LIN {X 0,Y 333.644,Z 264.427,A -85,B 0,C 180,E1 -14639.633,E2 -14639.633} C_VEL
LIN {X 0,Y 333.689,Z 264.417,A -85,B 0,C 180,E1 -14642.397,E2 -14642.397} C_VEL
LIN {X 0,Y 333.704,Z 264.416,A -85,B 0,C 180,E1 -14645.09,E2 -14645.09} C_VEL
LIN {X 0,Y 333.673,Z 264.443,A -85,B 0,C 180,E1 -14648.774,E2 -14648.774} C_VEL
LIN {X 0,Y 334.576,Z 267.116,A -85,B 0,C 180,E1 -14648.985,E2 -14648.985} C_VEL
LIN {X 0,Y 336.917,Z 269.949,A -85,B 0,C 180,E1 -14649.425,E2 -14649.425} C_VEL
LIN {X 0,Y 339.171,Z 273.256,A -85,B 0,C 180,E1 -14649.871,E2 -14649.871} C_VEL
LIN {X 0,Y 340.664,Z 274.981,A -85,B 0,C 180,E1 -14650.162,E2 -14650.162} C_VEL
LIN {X 0,Y 343.625,Z 278.711,A -85,B 0,C 180,E1 -14650.768,E2 -14650.768} C_VEL
LIN {X 0,Y 345.334,Z 280.75,A -85,B 0,C 180,E1 -14651.122,E2 -14651.122} C_VEL
LIN {X 0,Y 348.82,Z 284.693,A -85,B 0,C 180,E1 -14651.877,E2 -14651.877} C_VEL
LIN {X 0,Y 353.769,Z 290.158,A -85,B 0,C 180,E1 -14653.004,E2 -14653.004} C_VEL
LIN {X 0,Y 355.969,Z 292.267,A -85,B 0,C 180,E1 -14653.529,E2 -14653.529} C_VEL
LIN {X 0,Y 359.569,Z 296.096,A -85,B 0,C 180,E1 -14654.442,E2 -14654.442} C_VEL
LIN {X 0,Y 362.57,Z 298.711,A -85,B 0,C 180,E1 -14655.235,E2 -14655.235} C_VEL
LIN {X 0,Y 366.124,Z 302.39,A -85,B 0,C 180,E1 -14656.282,E2 -14656.282} C_VEL
LIN {X 0,Y 370.169,Z 305.771,A -85,B 0,C 180,E1 -14657.554,E2 -14657.554} C_VEL
LIN {X 0,Y 373.465,Z 309.144,A -85,B 0,C 180,E1 -14658.767,E2 -14658.767} C_VEL
LIN {X 0,Y 377.002,Z 311.663,A -85,B 0,C 180,E1 -14660.138,E2 -14660.138} C_VEL
LIN {X 0,Y 378.672,Z 312.756,A -85,B 0,C 180,E1 -14660.864,E2 -14660.864} C_VEL
LIN {X 0,Y 381.373,Z 315.868,A -85,B 0,C 180,E1 -14662.35,E2 -14662.35} C_VEL
LIN {X 0,Y 383.817,Z 317.899,A -85,B 0,C 180,E1 -14663.899,E2 -14663.899} C_VEL
LIN {X 0,Y 385.982,Z 319.066,A -85,B 0,C 180,E1 -14665.59,E2 -14665.59} C_VEL
LIN {X 0,Y 387.241,Z 319.408,A -85,B 0,C 180,E1 -14666.879,E2 -14666.879} C_VEL
LIN {X 0,Y 387.946,Z 319.576,A -85,B 0,C 180,E1 -14667.924,E2 -14667.924} C_VEL
LIN {X 0,Y 388.385,Z 319.645,A -85,B 0,C 180,E1 -14668.963,E2 -14668.963} C_VEL
LIN {X 0,Y 388.544,Z 319.673,A -85,B 0,C 180,E1 -14670,E2 -14670} C_VEL
LIN {X 0,Y 388.383,Z 319.645,A -85,B 0,C 180,E1 -14671.037,E2 -14671.037} C_VEL
LIN {X 0,Y 387.236,Z 319.4,A -85,B 0,C 180,E1 -14673.121,E2 -14673.121} C_VEL
LIN {X 0,Y 385.289,Z 318.79,A -85,B 0,C 180,E1 -14674.995,E2 -14674.995} C_VEL
LIN {X 0,Y 382.667,Z 317.06,A -85,B 0,C 180,E1 -14676.858,E2 -14676.858} C_VEL
LIN {X 0,Y 379.94,Z 314.347,A -85,B 0,C 180,E1 -14678.455,E2 -14678.455} C_VEL
LIN {X 0,Y 378.086,Z 312.243,A -85,B 0,C 180,E1 -14679.384,E2 -14679.384} C_VEL
LIN {X 0,Y 374.748,Z 310.2,A -85,B 0,C 180,E1 -14680.732,E2 -14680.732} C_VEL
LIN {X 0,Y 371.26,Z 307.035,A -85,B 0,C 180,E1 -14682.053,E2 -14682.053} C_VEL
LIN {X 0,Y 368.774,Z 304.446,A -85,B 0,C 180,E1 -14682.914,E2 -14682.914} C_VEL
LIN {X 0,Y 364.898,Z 301.318,A -85,B 0,C 180,E1 -14684.081,E2 -14684.081} C_VEL
LIN {X 0,Y 361.298,Z 297.476,A -85,B 0,C 180,E1 -14685.115,E2 -14685.115} C_VEL
LIN {X 0,Y 357.215,Z 293.734,A -85,B 0,C 180,E1 -14686.17,E2 -14686.17} C_VEL
LIN {X 0,Y 354.441,Z 290.752,A -85,B 0,C 180,E1 -14686.836,E2 -14686.836} C_VEL
LIN {X 0,Y 350.86,Z 287.08,A -85,B 0,C 180,E1 -14687.662,E2 -14687.662} C_VEL
LIN {X 0,Y 348.59,Z 284.464,A -85,B 0,C 180,E1 -14688.174,E2 -14688.174} C_VEL
LIN {X 0,Y 345.334,Z 280.748,A -85,B 0,C 180,E1 -14688.878,E2 -14688.878} C_VEL
LIN {X 0,Y 343.74,Z 278.843,A -85,B 0,C 180,E1 -14689.208,E2 -14689.208} C_VEL
LIN {X 0,Y 340.623,Z 274.921,A -85,B 0,C 180,E1 -14689.846,E2 -14689.846} C_VEL
LIN {X 0,Y 337.257,Z 270.639,A -85,B 0,C 180,E1 -14690.505,E2 -14690.505} C_VEL
LIN {X 0,Y 336.338,Z 269.129,A -85,B 0,C 180,E1 -14690.687,E2 -14690.687} C_VEL
LIN {X 0,Y 334.367,Z 266.73,A -85,B 0,C 180,E1 -14691.058,E2 -14691.058} C_VEL
LIN {X 0,Y 333.667,Z 264.421,A -85,B 0,C 180,E1 -14691.261,E2 -14691.261} C_VEL
LIN {X 0,Y 333.674,Z 264.419,A -85,B 0,C 180,E1 -14695.108,E2 -14695.108} C_VEL
LIN {X 0,Y 333.667,Z 264.421,A -85,B 0,C 180,E1 -14697.814,E2 -14697.814} C_VEL
LIN {X 0,Y 333.644,Z 264.427,A -85,B 0,C 180,E1 -14700.367,E2 -14700.367} C_VEL
LIN {X 0,Y 333.634,Z 264.424,A -85,B 0,C 180,E1 -14704.779,E2 -14704.779} C_VEL
LIN {X 0,Y 333.631,Z 264.424,A -85,B 0,C 180,E1 -14708.809,E2 -14708.809} C_VEL
LIN {X 0,Y 333.657,Z 264.421,A -85,B 0,C 180,E1 -14712.519,E2 -14712.519} C_VEL
LIN {X 0,Y 333.687,Z 264.421,A -85,B 0,C 180,E1 -14715.983,E2 -14715.983} C_VEL
LIN {X 0,Y 333.662,Z 264.421,A -85,B 0,C 180,E1 -14719.311,E2 -14719.311} C_VEL
LIN {X 0,Y 333.628,Z 264.425,A -85,B 0,C 180,E1 -14723.175,E2 -14723.175} C_VEL
LIN {X 0,Y 333.604,Z 264.427,A -85,B 0,C 180,E1 -14726.799,E2 -14726.799} C_VEL
LIN {X 0,Y 333.649,Z 264.423,A -85,B 0,C 180,E1 -14731.032,E2 -14731.032} C_VEL
LIN {X 0,Y 333.681,Z 264.417,A -85,B 0,C 180,E1 -14734.672,E2 -14734.672} C_VEL
LIN {X 0,Y 333.639,Z 264.423,A -85,B 0,C 180,E1 -14737.945,E2 -14737.945} C_VEL
LIN {X 0,Y 333.622,Z 264.423,A -85,B 0,C 180,E1 -14739.904,E2 -14739.904} C_VEL
LIN {X 0,Y 332.986,Z 264.507,A -85,B 0,C 180,E1 -14740.912,E2 -14740.912} C_VEL
LIN {X 0,Y 330.181,Z 264.858,A -85,B 0,C 180,E1 -14742.552,E2 -14742.552} C_VEL
LIN {X 0,Y 327.805,Z 265.156,A -85,B 0,C 180,E1 -14743.881,E2 -14743.881} C_VEL
LIN {X 0,Y 326.806,Z 265.278,A -85,B 0,C 180,E1 -14744.909,E2 -14744.909} C_VEL
LIN {X 0,Y 326.736,Z 265.285,A -85,B 0,C 180,E1 -14745.257,E2 -14745.257} C_VEL
LIN {X 0,Y 326.741,Z 265.286,A -85,B 0,C 180,E1 -14748.846,E2 -14748.846} C_VEL
LIN {X 0,Y 326.925,Z 265.261,A -85,B 0,C 180,E1 -14752.597,E2 -14752.597} C_VEL
LIN {X 0,Y 326.754,Z 265.282,A -85,B 0,C 180,E1 -14755.072,E2 -14755.072} C_VEL
LIN {X 0,Y 327.033,Z 265.241,A -85,B 0,C 180,E1 -14757.544,E2 -14757.544} C_VEL
LIN {X 0,Y 327.15,Z 265.228,A -85,B 0,C 180,E1 -14760.007,E2 -14760.007} C_VEL
LIN {X 0,Y 327.005,Z 265.252,A -85,B 0,C 180,E1 -14762.471,E2 -14762.471} C_VEL
LIN {X 0,Y 326.948,Z 265.258,A -85,B 0,C 180,E1 -14766.177,E2 -14766.177} C_VEL
LIN {X 0,Y 326.781,Z 265.278,A -85,B 0,C 180,E1 -14769.914,E2 -14769.914} C_VEL
LIN {X 0,Y 326.76,Z 265.28,A -85,B 0,C 180,E1 -14773.692,E2 -14773.692} C_VEL
LIN {X 0,Y 326.666,Z 265.292,A -85,B 0,C 180,E1 -14777.536,E2 -14777.536} C_VEL
LIN {X 0,Y 326.619,Z 265.298,A -85,B 0,C 180,E1 -14781.463,E2 -14781.463} C_VEL
LIN {X 0,Y 326.611,Z 265.3,A -85,B 0,C 180,E1 -14785.497,E2 -14785.497} C_VEL
LIN {X 0,Y 326.624,Z 265.3,A -85,B 0,C 180,E1 -14789.669,E2 -14789.669} C_VEL
LIN {X 0,Y 326.627,Z 265.299,A -85,B 0,C 180,E1 -14792.951,E2 -14792.951} C_VEL
LIN {X 0,Y 326.695,Z 265.648,A -85,B 0,C 180,E1 -14795.516,E2 -14795.516} C_VEL
LIN {X 0,Y 327.028,Z 268.288,A -85,B 0,C 180,E1 -14799.318,E2 -14799.318} C_VEL
LIN {X 0,Y 327.449,Z 271.2,A -85,B 0,C 180,E1 -14803.137,E2 -14803.137} C_VEL
LIN {X 0,Y 327.622,Z 272.801,A -85,B 0,C 180,E1 -14805.071,E2 -14805.071} C_VEL
LIN {X 0,Y 327.621,Z 275.669,A -85,B 0,C 180,E1 -14808.319,E2 -14808.319} C_VEL
LIN {X 0,Y 327.293,Z 278.686,A -85,B 0,C 180,E1 -14811.486,E2 -14811.486} C_VEL
LIN {X 0,Y 326.878,Z 282.026,A -85,B 0,C 180,E1 -14814.795,E2 -14814.795} C_VEL
LIN {X 0,Y 326.508,Z 284.828,A -85,B 0,C 180,E1 -14817.445,E2 -14817.445} C_VEL
LIN {X 0,Y 326.089,Z 287.929,A -85,B 0,C 180,E1 -14820.285,E2 -14820.285} C_VEL
LIN {X 0,Y 325.729,Z 291.054,A -85,B 0,C 180,E1 -14823.058,E2 -14823.058} C_VEL
LIN {X 0,Y 325.493,Z 294.197,A -85,B 0,C 180,E1 -14825.78,E2 -14825.78} C_VEL
LIN {X 0,Y 325.313,Z 296.391,A -85,B 0,C 180,E1 -14827.665,E2 -14827.665} C_VEL
LIN {X 0,Y 327.913,Z 307.333,A -85,B 0,C 180,E1 -14828.298,E2 -14828.298} C_VEL
LIN {X 0,Y 330.08,Z 318.555,A -85,B 0,C 180,E1 -14829.095,E2 -14829.095} C_VEL
LIN {X 0,Y 331.797,Z 331.19,A -85,B 0,C 180,E1 -14830.19,E2 -14830.19} C_VEL
LIN {X 0,Y 332.291,Z 337.754,A -85,B 0,C 180,E1 -14830.864,E2 -14830.864} C_VEL
LIN {X 0,Y 330.764,Z 349.942,A -85,B 0,C 180,E1 -14832.216,E2 -14832.216} C_VEL
LIN {X 0,Y 329.772,Z 357.691,A -85,B 0,C 180,E1 -14833.28,E2 -14833.28} C_VEL
LIN {X 0,Y 328.77,Z 365.484,A -85,B 0,C 180,E1 -14834.558,E2 -14834.558} C_VEL
LIN {X 0,Y 327.779,Z 373.031,A -85,B 0,C 180,E1 -14836.042,E2 -14836.042} C_VEL
LIN {X 0,Y 326.787,Z 379.566,A -85,B 0,C 180,E1 -14837.581,E2 -14837.581} C_VEL
LIN {X 0,Y 326.225,Z 384.069,A -85,B 0,C 180,E1 -14838.82,E2 -14838.82} C_VEL
LIN {X 0,Y 325.575,Z 389.562,A -85,B 0,C 180,E1 -14840.683,E2 -14840.683} C_VEL
LIN {X 0,Y 325.17,Z 393.888,A -85,B 0,C 180,E1 -14842.549,E2 -14842.549} C_VEL
LIN {X 0,Y 324.939,Z 396.93,A -85,B 0,C 180,E1 -14844.258,E2 -14844.258} C_VEL
LIN {X 0,Y 324.881,Z 399.445,A -85,B 0,C 180,E1 -14846.279,E2 -14846.279} C_VEL
LIN {X 0,Y 324.841,Z 400.504,A -85,B 0,C 180,E1 -14847.52,E2 -14847.52} C_VEL
LIN {X 0,Y 324.822,Z 401.092,A -85,B 0,C 180,E1 -14848.76,E2 -14848.76} C_VEL
LIN {X 0,Y 324.822,Z 401.092,A -85,B 0,C 180,E1 -14851.24,E2 -14851.24} C_VEL
LIN {X 0,Y 324.841,Z 400.504,A -85,B 0,C 180,E1 -14852.48,E2 -14852.48} C_VEL
LIN {X 0,Y 324.89,Z 398.056,A -85,B 0,C 180,E1 -14854.964,E2 -14854.964} C_VEL
LIN {X 0,Y 325.066,Z 395.106,A -85,B 0,C 180,E1 -14856.829,E2 -14856.829} C_VEL
LIN {X 0,Y 325.409,Z 391.116,A -85,B 0,C 180,E1 -14858.695,E2 -14858.695} C_VEL
LIN {X 0,Y 325.978,Z 385.985,A -85,B 0,C 180,E1 -14860.559,E2 -14860.559} C_VEL
LIN {X 0,Y 326.638,Z 380.722,A -85,B 0,C 180,E1 -14862.109,E2 -14862.109} C_VEL
LIN {X 0,Y 327.567,Z 374.407,A -85,B 0,C 180,E1 -14863.651,E2 -14863.651} C_VEL
LIN {X 0,Y 328.339,Z 368.454,A -85,B 0,C 180,E1 -14864.883,E2 -14864.883} C_VEL
LIN {X 0,Y 329.311,Z 361.139,A -85,B 0,C 180,E1 -14866.171,E2 -14866.171} C_VEL
LIN {X 0,Y 330.257,Z 353.344,A -85,B 0,C 180,E1 -14867.333,E2 -14867.333} C_VEL
LIN {X 0,Y 331.417,Z 344.836,A -85,B 0,C 180,E1 -14868.387,E2 -14868.387} C_VEL
LIN {X 0,Y 332.252,Z 337.753,A -85,B 0,C 180,E1 -14869.139,E2 -14869.139} C_VEL
LIN {X 0,Y 331.39,Z 327.713,A -85,B 0,C 180,E1 -14870.126,E2 -14870.126} C_VEL
LIN {X 0,Y 329.892,Z 317.576,A -85,B 0,C 180,E1 -14870.979,E2 -14870.979} C_VEL
LIN {X 0,Y 327.899,Z 307.287,A -85,B 0,C 180,E1 -14871.705,E2 -14871.705} C_VEL
LIN {X 0,Y 325.307,Z 296.391,A -85,B 0,C 180,E1 -14872.335,E2 -14872.335} C_VEL
LIN {X 0,Y 325.586,Z 292.61,A -85,B 0,C 180,E1 -14875.576,E2 -14875.576} C_VEL
LIN {X 0,Y 325.872,Z 289.477,A -85,B 0,C 180,E1 -14878.324,E2 -14878.324} C_VEL
LIN {X 0,Y 326.281,Z 286.366,A -85,B 0,C 180,E1 -14881.127,E2 -14881.127} C_VEL
LIN {X 0,Y 326.706,Z 283.278,A -85,B 0,C 180,E1 -14884.007,E2 -14884.007} C_VEL
LIN {X 0,Y 327.163,Z 279.83,A -85,B 0,C 180,E1 -14887.354,E2 -14887.354} C_VEL
LIN {X 0,Y 327.451,Z 277.155,A -85,B 0,C 180,E1 -14890.081,E2 -14890.081} C_VEL
LIN {X 0,Y 327.666,Z 274.144,A -85,B 0,C 180,E1 -14893.341,E2 -14893.341} C_VEL
LIN {X 0,Y 327.464,Z 271.387,A -85,B 0,C 180,E1 -14896.618,E2 -14896.618} C_VEL
LIN {X 0,Y 327.12,Z 268.859,A -85,B 0,C 180,E1 -14899.863,E2 -14899.863} C_VEL
LIN {X 0,Y 326.806,Z 266.661,A -85,B 0,C 180,E1 -14902.97,E2 -14902.97} C_VEL
LIN {X 0,Y 326.649,Z 265.423,A -85,B 0,C 180,E1 -14904.842,E2 -14904.842} C_VEL
LIN {X 0,Y 326.617,Z 265.303,A -85,B 0,C 180,E1 -14907.45,E2 -14907.45} C_VEL
LIN {X 0,Y 326.624,Z 265.3,A -85,B 0,C 180,E1 -14910.331,E2 -14910.331} C_VEL
LIN {X 0,Y 326.611,Z 265.299,A -85,B 0,C 180,E1 -14914.503,E2 -14914.503} C_VEL
LIN {X 0,Y 326.619,Z 265.298,A -85,B 0,C 180,E1 -14918.537,E2 -14918.537} C_VEL
LIN {X 0,Y 326.666,Z 265.292,A -85,B 0,C 180,E1 -14922.464,E2 -14922.464} C_VEL
LIN {X 0,Y 326.76,Z 265.28,A -85,B 0,C 180,E1 -14926.308,E2 -14926.308} C_VEL
LIN {X 0,Y 326.781,Z 265.278,A -85,B 0,C 180,E1 -14930.086,E2 -14930.086} C_VEL
LIN {X 0,Y 326.948,Z 265.258,A -85,B 0,C 180,E1 -14933.823,E2 -14933.823} C_VEL
LIN {X 0,Y 327.005,Z 265.252,A -85,B 0,C 180,E1 -14937.529,E2 -14937.529} C_VEL
LIN {X 0,Y 327.15,Z 265.228,A -85,B 0,C 180,E1 -14939.993,E2 -14939.993} C_VEL
LIN {X 0,Y 327.033,Z 265.241,A -85,B 0,C 180,E1 -14942.456,E2 -14942.456} C_VEL
LIN {X 0,Y 326.921,Z 265.258,A -85,B 0,C 180,E1 -14946.587,E2 -14946.587} C_VEL
LIN {X 0,Y 326.767,Z 265.277,A -85,B 0,C 180,E1 -14949.9,E2 -14949.9} C_VEL
LIN {X 0,Y 326.738,Z 265.282,A -85,B 0,C 180,E1 -14953.678,E2 -14953.678} C_VEL
LIN {X 0,Y 326.641,Z 265.295,A -85,B 0,C 180,E1 -14957.522,E2 -14957.522} C_VEL
LIN {X 0,Y 326.59,Z 265.301,A -85,B 0,C 180,E1 -14961.449,E2 -14961.449} C_VEL
LIN {X 0,Y 326.661,Z 265.291,A -85,B 0,C 180,E1 -14965.477,E2 -14965.477} C_VEL
LIN {X 0,Y 326.614,Z 265.301,A -85,B 0,C 180,E1 -14968.245,E2 -14968.245} C_VEL
LIN {X 0,Y 326.541,Z 265.307,A -85,B 0,C 180,E1 -14971.09,E2 -14971.09} C_VEL
LIN {X 0,Y 326.572,Z 265.305,A -85,B 0,C 180,E1 -14974.012,E2 -14974.012} C_VEL
LIN {X 0,Y 326.59,Z 265.301,A -85,B 0,C 180,E1 -14977.232,E2 -14977.232} C_VEL
LIN {X 0,Y 326.595,Z 265.305,A -85,B 0,C 180,E1 -14980.196,E2 -14980.196} C_VEL
LIN {X 0,Y 326.616,Z 265.298,A -85,B 0,C 180,E1 -14983.503,E2 -14983.503} C_VEL
LIN {X 0,Y 326.605,Z 265.299,A -85,B 0,C 180,E1 -14987.008,E2 -14987.008} C_VEL
LIN {X 0,Y 326.595,Z 265.3,A -85,B 0,C 180,E1 -14990.761,E2 -14990.761} C_VEL
LIN {X 0,Y 326.561,Z 265.306,A -85,B 0,C 180,E1 -14994.475,E2 -14994.475} C_VEL
LIN {X 0,Y 326.555,Z 265.308,A -85,B 0,C 180,E1 -14997.451,E2 -14997.451} C_VEL
LIN {X 0,Y 326.607,Z 265.3,A -85,B 0,C 180,E1 -15000.336,E2 -15000.336} C_VEL
LIN {X 0,Y 326.638,Z 265.296,A -85,B 0,C 180,E1 -15004.513,E2 -15004.513} C_VEL
LIN {X 0,Y 326.672,Z 265.295,A -85,B 0,C 180,E1 -15007.84,E2 -15007.84} C_VEL
LIN {X 0,Y 327.648,Z 268.131,A -85,B 0,C 180,E1 -15008.038,E2 -15008.038} C_VEL
LIN {X 0,Y 329.491,Z 270.627,A -85,B 0,C 180,E1 -15008.359,E2 -15008.359} C_VEL
LIN {X 0,Y 331.91,Z 274.081,A -85,B 0,C 180,E1 -15008.792,E2 -15008.792} C_VEL
LIN {X 0,Y 335.924,Z 279.255,A -85,B 0,C 180,E1 -15009.53,E2 -15009.53} C_VEL
LIN {X 0,Y 340.274,Z 284.52,A -85,B 0,C 180,E1 -15010.376,E2 -15010.376} C_VEL
LIN {X 0,Y 345.056,Z 290.05,A -85,B 0,C 180,E1 -15011.363,E2 -15011.363} C_VEL
LIN {X 0,Y 347.614,Z 292.874,A -85,B 0,C 180,E1 -15011.926,E2 -15011.926} C_VEL
LIN {X 0,Y 351.873,Z 297.157,A -85,B 0,C 180,E1 -15012.898,E2 -15012.898} C_VEL
LIN {X 0,Y 356.821,Z 302.359,A -85,B 0,C 180,E1 -15014.137,E2 -15014.137} C_VEL
LIN {X 0,Y 359.918,Z 305.126,A -85,B 0,C 180,E1 -15014.967,E2 -15014.967} C_VEL
LIN {X 0,Y 363.972,Z 309.216,A -85,B 0,C 180,E1 -15016.17,E2 -15016.17} C_VEL
LIN {X 0,Y 367.633,Z 312.25,A -85,B 0,C 180,E1 -15017.33,E2 -15017.33} C_VEL
LIN {X 0,Y 370.681,Z 315.425,A -85,B 0,C 180,E1 -15018.466,E2 -15018.466} C_VEL
LIN {X 0,Y 372.449,Z 316.832,A -85,B 0,C 180,E1 -15019.124,E2 -15019.124} C_VEL
LIN {X 0,Y 375.428,Z 318.686,A -85,B 0,C 180,E1 -15020.301,E2 -15020.301} C_VEL
LIN {X 0,Y 377.643,Z 321.068,A -85,B 0,C 180,E1 -15021.438,E2 -15021.438} C_VEL
LIN {X 0,Y 379.582,Z 323.003,A -85,B 0,C 180,E1 -15022.553,E2 -15022.553} C_VEL
LIN {X 0,Y 381.623,Z 324.651,A -85,B 0,C 180,E1 -15023.879,E2 -15023.879} C_VEL
LIN {X 0,Y 382.786,Z 325.372,A -85,B 0,C 180,E1 -15024.733,E2 -15024.733} C_VEL
LIN {X 0,Y 384.078,Z 325.881,A -85,B 0,C 180,E1 -15025.803,E2 -15025.803} C_VEL
LIN {X 0,Y 385.094,Z 326.177,A -85,B 0,C 180,E1 -15026.862,E2 -15026.862} C_VEL
LIN {X 0,Y 385.838,Z 326.343,A -85,B 0,C 180,E1 -15027.912,E2 -15027.912} C_VEL
LIN {X 0,Y 386.3,Z 326.425,A -85,B 0,C 180,E1 -15028.958,E2 -15028.958} C_VEL
LIN {X 0,Y 386.465,Z 326.455,A -85,B 0,C 180,E1 -15030,E2 -15030} C_VEL
LIN {X 0,Y 386.3,Z 326.423,A -85,B 0,C 180,E1 -15031.042,E2 -15031.042} C_VEL
LIN {X 0,Y 385.837,Z 326.335,A -85,B 0,C 180,E1 -15032.088,E2 -15032.088} C_VEL
LIN {X 0,Y 385.093,Z 326.165,A -85,B 0,C 180,E1 -15033.138,E2 -15033.138} C_VEL
LIN {X 0,Y 384.078,Z 325.904,A -85,B 0,C 180,E1 -15034.197,E2 -15034.197} C_VEL
LIN {X 0,Y 381.617,Z 324.646,A -85,B 0,C 180,E1 -15036.113,E2 -15036.113} C_VEL
LIN {X 0,Y 379.556,Z 323.023,A -85,B 0,C 180,E1 -15037.447,E2 -15037.447} C_VEL
LIN {X 0,Y 376.984,Z 320.257,A -85,B 0,C 180,E1 -15038.925,E2 -15038.925} C_VEL
LIN {X 0,Y 375.339,Z 318.691,A -85,B 0,C 180,E1 -15039.702,E2 -15039.702} C_VEL
LIN {X 0,Y 372.179,Z 316.641,A -85,B 0,C 180,E1 -15040.958,E2 -15040.958} C_VEL
LIN {X 0,Y 368.297,Z 313.039,A -85,B 0,C 180,E1 -15042.419,E2 -15042.419} C_VEL
LIN {X 0,Y 366.146,Z 310.865,A -85,B 0,C 180,E1 -15043.165,E2 -15043.165} C_VEL
LIN {X 0,Y 361.936,Z 307.355,A -85,B 0,C 180,E1 -15044.434,E2 -15044.434} C_VEL
LIN {X 0,Y 358.38,Z 303.659,A -85,B 0,C 180,E1 -15045.452,E2 -15045.452} C_VEL
LIN {X 0,Y 354.153,Z 299.731,A -85,B 0,C 180,E1 -15046.534,E2 -15046.534} C_VEL
LIN {X 0,Y 351.261,Z 296.662,A -85,B 0,C 180,E1 -15047.236,E2 -15047.236} C_VEL
LIN {X 0,Y 347.018,Z 292.065,A -85,B 0,C 180,E1 -15048.219,E2 -15048.219} C_VEL
LIN {X 0,Y 341.99,Z 286.597,A -85,B 0,C 180,E1 -15049.274,E2 -15049.274} C_VEL
LIN {X 0,Y 336.884,Z 280.409,A -85,B 0,C 180,E1 -15050.287,E2 -15050.287} C_VEL
LIN {X 0,Y 333.123,Z 275.646,A -85,B 0,C 180,E1 -15050.995,E2 -15050.995} C_VEL
LIN {X 0,Y 329.614,Z 270.891,A -85,B 0,C 180,E1 -15051.615,E2 -15051.615} C_VEL
LIN {X 0,Y 328.71,Z 269.451,A -85,B 0,C 180,E1 -15051.783,E2 -15051.783} C_VEL
LIN {X 0,Y 327.218,Z 267.323,A -85,B 0,C 180,E1 -15052.037,E2 -15052.037} C_VEL
LIN {X 0,Y 326.658,Z 265.297,A -85,B 0,C 180,E1 -15052.193,E2 -15052.193} C_VEL
LIN {X 0,Y 326.638,Z 265.296,A -85,B 0,C 180,E1 -15055.487,E2 -15055.487} C_VEL
LIN {X 0,Y 326.607,Z 265.3,A -85,B 0,C 180,E1 -15059.664,E2 -15059.664} C_VEL
LIN {X 0,Y 326.555,Z 265.31,A -85,B 0,C 180,E1 -15064.025,E2 -15064.025} C_VEL
LIN {X 0,Y 326.579,Z 265.302,A -85,B 0,C 180,E1 -15067.244,E2 -15067.244} C_VEL
LIN {X 0,Y 326.588,Z 265.305,A -85,B 0,C 180,E1 -15070.208,E2 -15070.208} C_VEL
LIN {X 0,Y 326.613,Z 265.3,A -85,B 0,C 180,E1 -15073.516,E2 -15073.516} C_VEL
LIN {X 0,Y 326.609,Z 265.298,A -85,B 0,C 180,E1 -15077.02,E2 -15077.02} C_VEL
LIN {X 0,Y 326.604,Z 265.299,A -85,B 0,C 180,E1 -15080.773,E2 -15080.773} C_VEL
LIN {X 0,Y 326.575,Z 265.303,A -85,B 0,C 180,E1 -15084.487,E2 -15084.487} C_VEL
LIN {X 0,Y 326.576,Z 265.307,A -85,B 0,C 180,E1 -15087.463,E2 -15087.463} C_VEL
LIN {X 0,Y 326.596,Z 265.3,A -85,B 0,C 180,E1 -15090.345,E2 -15090.345} C_VEL
LIN {X 0,Y 326.646,Z 265.297,A -85,B 0,C 180,E1 -15093.149,E2 -15093.149} C_VEL
LIN {X 0,Y 326.621,Z 265.298,A -85,B 0,C 180,E1 -15095.878,E2 -15095.878} C_VEL
LIN {X 0,Y 326.592,Z 265.3,A -85,B 0,C 180,E1 -15099.898,E2 -15099.898} C_VEL
LIN {X 0,Y 326.687,Z 265.289,A -85,B 0,C 180,E1 -15103.768,E2 -15103.768} C_VEL
LIN {X 0,Y 326.736,Z 265.285,A -85,B 0,C 180,E1 -15105.257,E2 -15105.257} C_VEL
LIN {X 0,Y 326.089,Z 265.364,A -85,B 0,C 180,E1 -15106.286,E2 -15106.286} C_VEL
LIN {X 0,Y 323.218,Z 265.721,A -85,B 0,C 180,E1 -15107.96,E2 -15107.96} C_VEL
LIN {X 0,Y 320.802,Z 266.023,A -85,B 0,C 180,E1 -15109.317,E2 -15109.317} C_VEL
LIN {X 0,Y 319.813,Z 266.144,A -85,B 0,C 180,E1 -15110.368,E2 -15110.368} C_VEL
LIN {X 0,Y 319.759,Z 266.151,A -85,B 0,C 180,E1 -15110.724,E2 -15110.724} C_VEL
LIN {X 0,Y 319.902,Z 266.134,A -85,B 0,C 180,E1 -15113.701,E2 -15113.701} C_VEL
LIN {X 0,Y 319.976,Z 266.119,A -85,B 0,C 180,E1 -15117.49,E2 -15117.49} C_VEL
LIN {X 0,Y 320.103,Z 266.105,A -85,B 0,C 180,E1 -15120.007,E2 -15120.007} C_VEL
LIN {X 0,Y 319.951,Z 266.131,A -85,B 0,C 180,E1 -15122.525,E2 -15122.525} C_VEL
LIN {X 0,Y 319.905,Z 266.136,A -85,B 0,C 180,E1 -15126.313,E2 -15126.313} C_VEL
LIN {X 0,Y 319.734,Z 266.157,A -85,B 0,C 180,E1 -15130.135,E2 -15130.135} C_VEL
LIN {X 0,Y 319.733,Z 266.157,A -85,B 0,C 180,E1 -15133.999,E2 -15133.999} C_VEL
LIN {X 0,Y 319.617,Z 266.172,A -85,B 0,C 180,E1 -15137.936,E2 -15137.936} C_VEL
LIN {X 0,Y 319.57,Z 266.179,A -85,B 0,C 180,E1 -15141.961,E2 -15141.961} C_VEL
LIN {X 0,Y 319.561,Z 266.182,A -85,B 0,C 180,E1 -15146.101,E2 -15146.101} C_VEL
LIN {X 0,Y 319.551,Z 266.179,A -85,B 0,C 180,E1 -15148.944,E2 -15148.944} C_VEL
LIN {X 0,Y 319.533,Z 266.186,A -85,B 0,C 180,E1 -15151.868,E2 -15151.868} C_VEL
LIN {X 0,Y 319.596,Z 266.369,A -85,B 0,C 180,E1 -15154.879,E2 -15154.879} C_VEL
LIN {X 0,Y 319.875,Z 268.411,A -85,B 0,C 180,E1 -15157.972,E2 -15157.972} C_VEL
LIN {X 0,Y 320.29,Z 271.147,A -85,B 0,C 180,E1 -15161.752,E2 -15161.752} C_VEL
LIN {X 0,Y 320.546,Z 273.352,A -85,B 0,C 180,E1 -15164.563,E2 -15164.563} C_VEL
LIN {X 0,Y 320.603,Z 275.585,A -85,B 0,C 180,E1 -15167.192,E2 -15167.192} C_VEL
LIN {X 0,Y 320.398,Z 278.277,A -85,B 0,C 180,E1 -15170.158,E2 -15170.158} C_VEL
LIN {X 0,Y 319.968,Z 281.638,A -85,B 0,C 180,E1 -15173.627,E2 -15173.627} C_VEL
LIN {X 0,Y 319.521,Z 284.771,A -85,B 0,C 180,E1 -15176.71,E2 -15176.71} C_VEL
LIN {X 0,Y 319.17,Z 287.804,A -85,B 0,C 180,E1 -15179.573,E2 -15179.573} C_VEL
LIN {X 0,Y 318.558,Z 292.471,A -85,B 0,C 180,E1 -15183.818,E2 -15183.818} C_VEL
LIN {X 0,Y 318.271,Z 296.223,A -85,B 0,C 180,E1 -15187.143,E2 -15187.143} C_VEL
LIN {X 0,Y 320.641,Z 305.995,A -85,B 0,C 180,E1 -15187.725,E2 -15187.725} C_VEL
LIN {X 0,Y 322.656,Z 315.519,A -85,B 0,C 180,E1 -15188.408,E2 -15188.408} C_VEL
LIN {X 0,Y 324.097,Z 324.777,A -85,B 0,C 180,E1 -15189.177,E2 -15189.177} C_VEL
LIN {X 0,Y 325.018,Z 332.631,A -85,B 0,C 180,E1 -15189.924,E2 -15189.924} C_VEL
LIN {X 0,Y 325.421,Z 339.17,A -85,B 0,C 180,E1 -15190.607,E2 -15190.607} C_VEL
LIN {X 0,Y 323.991,Z 349.747,A -85,B 0,C 180,E1 -15191.831,E2 -15191.831} C_VEL
LIN {X 0,Y 322.927,Z 357.491,A -85,B 0,C 180,E1 -15192.914,E2 -15192.914} C_VEL
LIN {X 0,Y 321.844,Z 365.63,A -85,B 0,C 180,E1 -15194.285,E2 -15194.285} C_VEL
LIN {X 0,Y 320.875,Z 372.836,A -85,B 0,C 180,E1 -15195.736,E2 -15195.736} C_VEL
LIN {X 0,Y 319.84,Z 379.371,A -85,B 0,C 180,E1 -15197.307,E2 -15197.307} C_VEL
LIN {X 0,Y 319.215,Z 383.873,A -85,B 0,C 180,E1 -15198.572,E2 -15198.572} C_VEL
LIN {X 0,Y 318.53,Z 389.366,A -85,B 0,C 180,E1 -15200.475,E2 -15200.475} C_VEL
LIN {X 0,Y 318.094,Z 393.693,A -85,B 0,C 180,E1 -15202.382,E2 -15202.382} C_VEL
LIN {X 0,Y 317.853,Z 396.977,A -85,B 0,C 180,E1 -15204.301,E2 -15204.301} C_VEL
LIN {X 0,Y 317.791,Z 399.25,A -85,B 0,C 180,E1 -15206.196,E2 -15206.196} C_VEL
LIN {X 0,Y 317.762,Z 400.309,A -85,B 0,C 180,E1 -15207.465,E2 -15207.465} C_VEL
LIN {X 0,Y 317.735,Z 400.898,A -85,B 0,C 180,E1 -15208.733,E2 -15208.733} C_VEL
LIN {X 0,Y 317.735,Z 400.898,A -85,B 0,C 180,E1 -15211.267,E2 -15211.267} C_VEL
LIN {X 0,Y 317.762,Z 400.309,A -85,B 0,C 180,E1 -15212.535,E2 -15212.535} C_VEL
LIN {X 0,Y 317.806,Z 397.861,A -85,B 0,C 180,E1 -15215.075,E2 -15215.075} C_VEL
LIN {X 0,Y 318.004,Z 394.911,A -85,B 0,C 180,E1 -15216.982,E2 -15216.982} C_VEL
LIN {X 0,Y 318.37,Z 390.921,A -85,B 0,C 180,E1 -15218.889,E2 -15218.889} C_VEL
LIN {X 0,Y 318.968,Z 385.79,A -85,B 0,C 180,E1 -15220.794,E2 -15220.794} C_VEL
LIN {X 0,Y 319.65,Z 380.526,A -85,B 0,C 180,E1 -15222.378,E2 -15222.378} C_VEL
LIN {X 0,Y 320.644,Z 374.212,A -85,B 0,C 180,E1 -15223.951,E2 -15223.951} C_VEL
LIN {X 0,Y 321.674,Z 366.94,A -85,B 0,C 180,E1 -15225.462,E2 -15225.462} C_VEL
LIN {X 0,Y 322.64,Z 359.411,A -85,B 0,C 180,E1 -15226.775,E2 -15226.775} C_VEL
LIN {X 0,Y 323.816,Z 350.881,A -85,B 0,C 180,E1 -15228.015,E2 -15228.015} C_VEL
LIN {X 0,Y 325.212,Z 340.587,A -85,B 0,C 180,E1 -15229.242,E2 -15229.242} C_VEL
LIN {X 0,Y 325.335,Z 335.915,A -85,B 0,C 180,E1 -15229.726,E2 -15229.726} C_VEL
LIN {X 0,Y 324.319,Z 326.334,A -85,B 0,C 180,E1 -15230.681,E2 -15230.681} C_VEL
LIN {X 0,Y 322.827,Z 316.618,A -85,B 0,C 180,E1 -15231.509,E2 -15231.509} C_VEL
LIN {X 0,Y 320.819,Z 306.71,A -85,B 0,C 180,E1 -15232.227,E2 -15232.227} C_VEL
LIN {X 0,Y 318.304,Z 296.823,A -85,B 0,C 180,E1 -15232.83,E2 -15232.83} C_VEL
LIN {X 0,Y 318.264,Z 296.224,A -85,B 0,C 180,E1 -15232.856,E2 -15232.856} C_VEL
LIN {X 0,Y 318.554,Z 292.458,A -85,B 0,C 180,E1 -15236.183,E2 -15236.183} C_VEL
LIN {X 0,Y 319.171,Z 287.781,A -85,B 0,C 180,E1 -15240.427,E2 -15240.427} C_VEL
LIN {X 0,Y 319.75,Z 283.162,A -85,B 0,C 180,E1 -15244.852,E2 -15244.852} C_VEL
LIN {X 0,Y 320.178,Z 280.103,A -85,B 0,C 180,E1 -15247.922,E2 -15247.922} C_VEL
LIN {X 0,Y 320.579,Z 276.455,A -85,B 0,C 180,E1 -15251.801,E2 -15251.801} C_VEL
LIN {X 0,Y 320.591,Z 274.074,A -85,B 0,C 180,E1 -15254.546,E2 -15254.546} C_VEL
LIN {X 0,Y 320.278,Z 271.133,A -85,B 0,C 180,E1 -15258.25,E2 -15258.25} C_VEL
LIN {X 0,Y 319.876,Z 268.408,A -85,B 0,C 180,E1 -15262.028,E2 -15262.028} C_VEL
LIN {X 0,Y 319.597,Z 266.372,A -85,B 0,C 180,E1 -15265.122,E2 -15265.122} C_VEL
LIN {X 0,Y 319.533,Z 266.187,A -85,B 0,C 180,E1 -15268.132,E2 -15268.132} C_VEL
LIN {X 0,Y 319.579,Z 266.178,A -85,B 0,C 180,E1 -15271.598,E2 -15271.598} C_VEL
LIN {X 0,Y 319.559,Z 266.178,A -85,B 0,C 180,E1 -15275.294,E2 -15275.294} C_VEL
LIN {X 0,Y 319.57,Z 266.179,A -85,B 0,C 180,E1 -15278.039,E2 -15278.039} C_VEL
LIN {X 0,Y 319.617,Z 266.172,A -85,B 0,C 180,E1 -15282.064,E2 -15282.064} C_VEL
LIN {X 0,Y 319.733,Z 266.157,A -85,B 0,C 180,E1 -15286.001,E2 -15286.001} C_VEL
LIN {X 0,Y 319.734,Z 266.157,A -85,B 0,C 180,E1 -15289.865,E2 -15289.865} C_VEL
LIN {X 0,Y 319.905,Z 266.136,A -85,B 0,C 180,E1 -15293.687,E2 -15293.687} C_VEL
LIN {X 0,Y 319.951,Z 266.131,A -85,B 0,C 180,E1 -15297.475,E2 -15297.475} C_VEL
LIN {X 0,Y 320.103,Z 266.105,A -85,B 0,C 180,E1 -15299.993,E2 -15299.993} C_VEL
LIN {X 0,Y 319.976,Z 266.119,A -85,B 0,C 180,E1 -15302.51,E2 -15302.51} C_VEL
LIN {X 0,Y 319.884,Z 266.135,A -85,B 0,C 180,E1 -15306.575,E2 -15306.575} C_VEL
LIN {X 0,Y 319.719,Z 266.155,A -85,B 0,C 180,E1 -15310.12,E2 -15310.12} C_VEL
LIN {X 0,Y 319.712,Z 266.157,A -85,B 0,C 180,E1 -15313.985,E2 -15313.985} C_VEL
LIN {X 0,Y 319.591,Z 266.173,A -85,B 0,C 180,E1 -15317.922,E2 -15317.922} C_VEL
LIN {X 0,Y 319.541,Z 266.179,A -85,B 0,C 180,E1 -15321.947,E2 -15321.947} C_VEL
LIN {X 0,Y 319.587,Z 266.174,A -85,B 0,C 180,E1 -15326.082,E2 -15326.082} C_VEL
LIN {X 0,Y 319.536,Z 266.181,A -85,B 0,C 180,E1 -15328.928,E2 -15328.928} C_VEL
LIN {X 0,Y 319.492,Z 266.186,A -85,B 0,C 180,E1 -15331.855,E2 -15331.855} C_VEL
LIN {X 0,Y 319.543,Z 266.179,A -85,B 0,C 180,E1 -15335.536,E2 -15335.536} C_VEL
LIN {X 0,Y 319.544,Z 266.181,A -85,B 0,C 180,E1 -15338,E2 -15338} C_VEL
LIN {X 0,Y 319.561,Z 266.177,A -85,B 0,C 180,E1 -15341.606,E2 -15341.606} C_VEL
LIN {X 0,Y 319.602,Z 266.171,A -85,B 0,C 180,E1 -15345.279,E2 -15345.279} C_VEL
LIN {X 0,Y 319.537,Z 266.18,A -85,B 0,C 180,E1 -15348.714,E2 -15348.714} C_VEL
LIN {X 0,Y 319.533,Z 266.182,A -85,B 0,C 180,E1 -15352.338,E2 -15352.338} C_VEL
LIN {X 0,Y 319.509,Z 266.184,A -85,B 0,C 180,E1 -15355.118,E2 -15355.118} C_VEL
LIN {X 0,Y 319.517,Z 266.183,A -85,B 0,C 180,E1 -15359.054,E2 -15359.054} C_VEL
LIN {X 0,Y 319.555,Z 266.178,A -85,B 0,C 180,E1 -15362.494,E2 -15362.494} C_VEL
LIN {X 0,Y 319.573,Z 266.179,A -85,B 0,C 180,E1 -15365.302,E2 -15365.302} C_VEL
LIN {X 0,Y 319.596,Z 266.175,A -85,B 0,C 180,E1 -15367.036,E2 -15367.036} C_VEL
LIN {X 0,Y 320.559,Z 268.949,A -85,B 0,C 180,E1 -15367.213,E2 -15367.213} C_VEL
LIN {X 0,Y 322.303,Z 271.645,A -85,B 0,C 180,E1 -15367.478,E2 -15367.478} C_VEL
LIN {X 0,Y 327.533,Z 279.089,A -85,B 0,C 180,E1 -15368.33,E2 -15368.33} C_VEL
LIN {X 0,Y 332.283,Z 284.992,A -85,B 0,C 180,E1 -15369.177,E2 -15369.177} C_VEL
LIN {X 0,Y 336.512,Z 290.097,A -85,B 0,C 180,E1 -15369.991,E2 -15369.991} C_VEL
LIN {X 0,Y 341.572,Z 295.882,A -85,B 0,C 180,E1 -15371.031,E2 -15371.031} C_VEL
LIN {X 0,Y 347.201,Z 301.98,A -85,B 0,C 180,E1 -15372.304,E2 -15372.304} C_VEL
LIN {X 0,Y 350.341,Z 305.169,A -85,B 0,C 180,E1 -15373.055,E2 -15373.055} C_VEL
LIN {X 0,Y 354.65,Z 309.396,A -85,B 0,C 180,E1 -15374.167,E2 -15374.167} C_VEL
LIN {X 0,Y 356.859,Z 311.452,A -85,B 0,C 180,E1 -15374.76,E2 -15374.76} C_VEL
LIN {X 0,Y 361.736,Z 316.176,A -85,B 0,C 180,E1 -15376.228,E2 -15376.228} C_VEL
LIN {X 0,Y 364.843,Z 318.849,A -85,B 0,C 180,E1 -15377.224,E2 -15377.224} C_VEL
LIN {X 0,Y 367.926,Z 321.958,A -85,B 0,C 180,E1 -15378.378,E2 -15378.378} C_VEL
LIN {X 0,Y 371.38,Z 324.402,A -85,B 0,C 180,E1 -15379.697,E2 -15379.697} C_VEL
LIN {X 0,Y 373.644,Z 326.232,A -85,B 0,C 180,E1 -15380.702,E2 -15380.702} C_VEL
LIN {X 0,Y 376.79,Z 329.513,A -85,B 0,C 180,E1 -15382.498,E2 -15382.498} C_VEL
LIN {X 0,Y 378.513,Z 330.922,A -85,B 0,C 180,E1 -15383.604,E2 -15383.604} C_VEL
LIN {X 0,Y 380.753,Z 332.189,A -85,B 0,C 180,E1 -15385.254,E2 -15385.254} C_VEL
LIN {X 0,Y 382.42,Z 332.747,A -85,B 0,C 180,E1 -15386.84,E2 -15386.84} C_VEL
LIN {X 0,Y 383.196,Z 332.918,A -85,B 0,C 180,E1 -15387.898,E2 -15387.898} C_VEL
LIN {X 0,Y 383.675,Z 332.999,A -85,B 0,C 180,E1 -15388.95,E2 -15388.95} C_VEL
LIN {X 0,Y 383.839,Z 333.034,A -85,B 0,C 180,E1 -15390,E2 -15390} C_VEL
LIN {X 0,Y 383.675,Z 333,A -85,B 0,C 180,E1 -15391.05,E2 -15391.05} C_VEL
LIN {X 0,Y 383.196,Z 332.914,A -85,B 0,C 180,E1 -15392.102,E2 -15392.102} C_VEL
LIN {X 0,Y 382.418,Z 332.745,A -85,B 0,C 180,E1 -15393.16,E2 -15393.16} C_VEL
LIN {X 0,Y 380.752,Z 332.195,A -85,B 0,C 180,E1 -15394.744,E2 -15394.744} C_VEL
LIN {X 0,Y 378.498,Z 330.934,A -85,B 0,C 180,E1 -15396.396,E2 -15396.396} C_VEL
LIN {X 0,Y 376.043,Z 328.77,A -85,B 0,C 180,E1 -15397.96,E2 -15397.96} C_VEL
LIN {X 0,Y 372.625,Z 325.266,A -85,B 0,C 180,E1 -15399.773,E2 -15399.773} C_VEL
LIN {X 0,Y 369.678,Z 323.324,A -85,B 0,C 180,E1 -15400.959,E2 -15400.959} C_VEL
LIN {X 0,Y 366.469,Z 320.528,A -85,B 0,C 180,E1 -15402.178,E2 -15402.178} C_VEL
LIN {X 0,Y 361.724,Z 316.186,A -85,B 0,C 180,E1 -15403.764,E2 -15403.764} C_VEL
LIN {X 0,Y 358.371,Z 313.178,A -85,B 0,C 180,E1 -15404.77,E2 -15404.77} C_VEL
LIN {X 0,Y 355.406,Z 309.993,A -85,B 0,C 180,E1 -15405.638,E2 -15405.638} C_VEL
LIN {X 0,Y 350.616,Z 305.528,A -85,B 0,C 180,E1 -15406.869,E2 -15406.869} C_VEL
LIN {X 0,Y 347.512,Z 302.275,A -85,B 0,C 180,E1 -15407.626,E2 -15407.626} C_VEL
LIN {X 0,Y 343.168,Z 297.499,A -85,B 0,C 180,E1 -15408.629,E2 -15408.629} C_VEL
LIN {X 0,Y 338.455,Z 292.464,A -85,B 0,C 180,E1 -15409.612,E2 -15409.612} C_VEL
LIN {X 0,Y 332.78,Z 285.598,A -85,B 0,C 180,E1 -15410.73,E2 -15410.73} C_VEL
LIN {X 0,Y 328.806,Z 280.649,A -85,B 0,C 180,E1 -15411.451,E2 -15411.451} C_VEL
LIN {X 0,Y 325.11,Z 275.753,A -85,B 0,C 180,E1 -15412.076,E2 -15412.076} C_VEL
LIN {X 0,Y 322.163,Z 271.336,A -85,B 0,C 180,E1 -15412.547,E2 -15412.547} C_VEL
LIN {X 0,Y 319.937,Z 267.586,A -85,B 0,C 180,E1 -15412.886,E2 -15412.886} C_VEL
LIN {X 0,Y 319.591,Z 266.175,A -85,B 0,C 180,E1 -15412.972,E2 -15412.972} C_VEL
LIN {X 0,Y 319.582,Z 266.178,A -85,B 0,C 180,E1 -15416.092,E2 -15416.092} C_VEL
LIN {X 0,Y 319.536,Z 266.181,A -85,B 0,C 180,E1 -15418.938,E2 -15418.938} C_VEL
LIN {X 0,Y 319.48,Z 266.19,A -85,B 0,C 180,E1 -15421.867,E2 -15421.867} C_VEL
LIN {X 0,Y 319.529,Z 266.182,A -85,B 0,C 180,E1 -15425.548,E2 -15425.548} C_VEL
LIN {X 0,Y 319.55,Z 266.183,A -85,B 0,C 180,E1 -15428.01,E2 -15428.01} C_VEL
LIN {X 0,Y 319.556,Z 266.179,A -85,B 0,C 180,E1 -15431.618,E2 -15431.618} C_VEL
LIN {X 0,Y 319.603,Z 266.172,A -85,B 0,C 180,E1 -15435.291,E2 -15435.291} C_VEL
LIN {X 0,Y 319.543,Z 266.179,A -85,B 0,C 180,E1 -15438.727,E2 -15438.727} C_VEL
LIN {X 0,Y 319.544,Z 266.179,A -85,B 0,C 180,E1 -15442.35,E2 -15442.35} C_VEL
LIN {X 0,Y 319.524,Z 266.182,A -85,B 0,C 180,E1 -15445.13,E2 -15445.13} C_VEL
LIN {X 0,Y 319.492,Z 266.186,A -85,B 0,C 180,E1 -15448.145,E2 -15448.145} C_VEL
LIN {X 0,Y 319.576,Z 266.179,A -85,B 0,C 180,E1 -15451.6,E2 -15451.6} C_VEL
LIN {X 0,Y 319.575,Z 266.178,A -85,B 0,C 180,E1 -15455.311,E2 -15455.311} C_VEL
LIN {X 0,Y 319.553,Z 266.18,A -85,B 0,C 180,E1 -15459.406,E2 -15459.406} C_VEL
LIN {X 0,Y 319.63,Z 266.171,A -85,B 0,C 180,E1 -15463.399,E2 -15463.399} C_VEL
LIN {X 0,Y 319.712,Z 266.157,A -85,B 0,C 180,E1 -15466.015,E2 -15466.015} C_VEL
LIN {X 0,Y 319.719,Z 266.155,A -85,B 0,C 180,E1 -15469.88,E2 -15469.88} C_VEL
LIN {X 0,Y 319.759,Z 266.151,A -85,B 0,C 180,E1 -15470.724,E2 -15470.724} C_VEL
LIN {X 0,Y 319.482,Z 266.19,A -85,B 0,C 180,E1 -15471.427,E2 -15471.427} C_VEL
LIN {X 0,Y 317.513,Z 266.441,A -85,B 0,C 180,E1 -15472.806,E2 -15472.806} C_VEL
LIN {X 0,Y 313.718,Z 266.911,A -85,B 0,C 180,E1 -15474.871,E2 -15474.871} C_VEL
LIN {X 0,Y 312.733,Z 267.026,A -85,B 0,C 180,E1 -15475.947,E2 -15475.947} C_VEL
LIN {X 0,Y 312.696,Z 267.027,A -85,B 0,C 180,E1 -15476.311,E2 -15476.311} C_VEL
LIN {X 0,Y 312.977,Z 266.992,A -85,B 0,C 180,E1 -15478.721,E2 -15478.721} C_VEL
LIN {X 0,Y 312.976,Z 266.997,A -85,B 0,C 180,E1 -15481.294,E2 -15481.294} C_VEL
LIN {X 0,Y 312.849,Z 267.017,A -85,B 0,C 180,E1 -15486.456,E2 -15486.456} C_VEL
LIN {X 0,Y 312.749,Z 267.027,A -85,B 0,C 180,E1 -15489.057,E2 -15489.057} C_VEL
LIN {X 0,Y 312.634,Z 267.041,A -85,B 0,C 180,E1 -15492.998,E2 -15492.998} C_VEL
LIN {X 0,Y 312.624,Z 267.042,A -85,B 0,C 180,E1 -15495.657,E2 -15495.657} C_VEL
LIN {X 0,Y 312.542,Z 267.052,A -85,B 0,C 180,E1 -15499.719,E2 -15499.719} C_VEL
LIN {X 0,Y 312.525,Z 267.054,A -85,B 0,C 180,E1 -15502.783,E2 -15502.783} C_VEL
LIN {X 0,Y 312.518,Z 267.059,A -85,B 0,C 180,E1 -15505.906,E2 -15505.906} C_VEL
LIN {X 0,Y 312.504,Z 267.059,A -85,B 0,C 180,E1 -15509.661,E2 -15509.661} C_VEL
LIN {X 0,Y 312.534,Z 267.059,A -85,B 0,C 180,E1 -15513.695,E2 -15513.695} C_VEL
LIN {X 0,Y 312.53,Z 267.09,A -85,B 0,C 180,E1 -15514.214,E2 -15514.214} C_VEL
LIN {X 0,Y 312.865,Z 269.636,A -85,B 0,C 180,E1 -15518.168,E2 -15518.168} C_VEL
LIN {X 0,Y 313.131,Z 271.336,A -85,B 0,C 180,E1 -15520.615,E2 -15520.615} C_VEL
LIN {X 0,Y 313.474,Z 274.031,A -85,B 0,C 180,E1 -15524.159,E2 -15524.159} C_VEL
LIN {X 0,Y 313.572,Z 276.979,A -85,B 0,C 180,E1 -15527.706,E2 -15527.706} C_VEL
LIN {X 0,Y 313.225,Z 280.021,A -85,B 0,C 180,E1 -15531.08,E2 -15531.08} C_VEL
LIN {X 0,Y 312.814,Z 283.049,A -85,B 0,C 180,E1 -15534.259,E2 -15534.259} C_VEL
LIN {X 0,Y 312.34,Z 286.116,A -85,B 0,C 180,E1 -15537.316,E2 -15537.316} C_VEL
LIN {X 0,Y 311.92,Z 289.206,A -85,B 0,C 180,E1 -15540.286,E2 -15540.286} C_VEL
LIN {X 0,Y 311.43,Z 293.867,A -85,B 0,C 180,E1 -15544.611,E2 -15544.611} C_VEL
LIN {X 0,Y 311.227,Z 296.188,A -85,B 0,C 180,E1 -15546.606,E2 -15546.606} C_VEL
LIN {X 0,Y 313.735,Z 306.221,A -85,B 0,C 180,E1 -15547.229,E2 -15547.229} C_VEL
LIN {X 0,Y 315.892,Z 316.453,A -85,B 0,C 180,E1 -15547.997,E2 -15547.997} C_VEL
LIN {X 0,Y 317.496,Z 327.102,A -85,B 0,C 180,E1 -15548.935,E2 -15548.935} C_VEL
LIN {X 0,Y 318.556,Z 337.354,A -85,B 0,C 180,E1 -15550.004,E2 -15550.004} C_VEL
LIN {X 0,Y 318.207,Z 343.097,A -85,B 0,C 180,E1 -15550.653,E2 -15550.653} C_VEL
LIN {X 0,Y 316.9,Z 351.821,A -85,B 0,C 180,E1 -15551.745,E2 -15551.745} C_VEL
LIN {X 0,Y 315.857,Z 359.216,A -85,B 0,C 180,E1 -15552.854,E2 -15552.854} C_VEL
LIN {X 0,Y 314.766,Z 366.892,A -85,B 0,C 180,E1 -15554.22,E2 -15554.22} C_VEL
LIN {X 0,Y 313.719,Z 374.016,A -85,B 0,C 180,E1 -15555.734,E2 -15555.734} C_VEL
LIN {X 0,Y 312.689,Z 380.331,A -85,B 0,C 180,E1 -15557.342,E2 -15557.342} C_VEL
LIN {X 0,Y 311.968,Z 385.594,A -85,B 0,C 180,E1 -15558.961,E2 -15558.961} C_VEL
LIN {X 0,Y 311.313,Z 390.725,A -85,B 0,C 180,E1 -15560.908,E2 -15560.908} C_VEL
LIN {X 0,Y 310.939,Z 394.715,A -85,B 0,C 180,E1 -15562.859,E2 -15562.859} C_VEL
LIN {X 0,Y 310.717,Z 397.666,A -85,B 0,C 180,E1 -15564.809,E2 -15564.809} C_VEL
LIN {X 0,Y 310.686,Z 400.115,A -85,B 0,C 180,E1 -15567.407,E2 -15567.407} C_VEL
LIN {X 0,Y 310.651,Z 400.704,A -85,B 0,C 180,E1 -15568.704,E2 -15568.704} C_VEL
LIN {X 0,Y 310.651,Z 400.704,A -85,B 0,C 180,E1 -15571.296,E2 -15571.296} C_VEL
LIN {X 0,Y 310.685,Z 400.115,A -85,B 0,C 180,E1 -15572.593,E2 -15572.593} C_VEL
LIN {X 0,Y 310.71,Z 397.665,A -85,B 0,C 180,E1 -15575.191,E2 -15575.191} C_VEL
LIN {X 0,Y 310.937,Z 394.715,A -85,B 0,C 180,E1 -15577.141,E2 -15577.141} C_VEL
LIN {X 0,Y 311.313,Z 390.725,A -85,B 0,C 180,E1 -15579.092,E2 -15579.092} C_VEL
LIN {X 0,Y 311.968,Z 385.594,A -85,B 0,C 180,E1 -15581.039,E2 -15581.039} C_VEL
LIN {X 0,Y 312.689,Z 380.331,A -85,B 0,C 180,E1 -15582.658,E2 -15582.658} C_VEL
LIN {X 0,Y 313.718,Z 374.016,A -85,B 0,C 180,E1 -15584.266,E2 -15584.266} C_VEL
LIN {X 0,Y 314.796,Z 366.915,A -85,B 0,C 180,E1 -15585.774,E2 -15585.774} C_VEL
LIN {X 0,Y 315.815,Z 359.215,A -85,B 0,C 180,E1 -15587.149,E2 -15587.149} C_VEL
LIN {X 0,Y 317.038,Z 350.685,A -85,B 0,C 180,E1 -15588.414,E2 -15588.414} C_VEL
LIN {X 0,Y 318.504,Z 340.392,A -85,B 0,C 180,E1 -15589.663,E2 -15589.663} C_VEL
LIN {X 0,Y 318.255,Z 334.071,A -85,B 0,C 180,E1 -15590.353,E2 -15590.353} C_VEL
LIN {X 0,Y 317.192,Z 324.76,A -85,B 0,C 180,E1 -15591.283,E2 -15591.283} C_VEL
LIN {X 0,Y 315.721,Z 315.475,A -85,B 0,C 180,E1 -15592.081,E2 -15592.081} C_VEL
LIN {X 0,Y 313.59,Z 305.714,A -85,B 0,C 180,E1 -15592.807,E2 -15592.807} C_VEL
LIN {X 0,Y 311.222,Z 296.026,A -85,B 0,C 180,E1 -15593.431,E2 -15593.431} C_VEL
LIN {X 0,Y 311.54,Z 292.299,A -85,B 0,C 180,E1 -15596.819,E2 -15596.819} C_VEL
LIN {X 0,Y 312.155,Z 287.654,A -85,B 0,C 180,E1 -15601.186,E2 -15601.186} C_VEL
LIN {X 0,Y 312.584,Z 284.574,A -85,B 0,C 180,E1 -15604.199,E2 -15604.199} C_VEL
LIN {X 0,Y 313.04,Z 281.507,A -85,B 0,C 180,E1 -15607.312,E2 -15607.312} C_VEL
LIN {X 0,Y 313.413,Z 278.485,A -85,B 0,C 180,E1 -15610.563,E2 -15610.563} C_VEL
LIN {X 0,Y 313.539,Z 276.94,A -85,B 0,C 180,E1 -15612.287,E2 -15612.287} C_VEL
LIN {X 0,Y 313.559,Z 275.363,A -85,B 0,C 180,E1 -15614.166,E2 -15614.166} C_VEL
LIN {X 0,Y 313.307,Z 272.524,A -85,B 0,C 180,E1 -15617.751,E2 -15617.751} C_VEL
LIN {X 0,Y 312.952,Z 270.177,A -85,B 0,C 180,E1 -15621.032,E2 -15621.032} C_VEL
LIN {X 0,Y 312.676,Z 268.055,A -85,B 0,C 180,E1 -15624.233,E2 -15624.233} C_VEL
LIN {X 0,Y 312.53,Z 267.087,A -85,B 0,C 180,E1 -15625.786,E2 -15625.786} C_VEL
LIN {X 0,Y 312.515,Z 267.058,A -85,B 0,C 180,E1 -15628.846,E2 -15628.846} C_VEL
LIN {X 0,Y 312.536,Z 267.057,A -85,B 0,C 180,E1 -15631.814,E2 -15631.814} C_VEL
LIN {X 0,Y 312.533,Z 267.053,A -85,B 0,C 180,E1 -15634.7,E2 -15634.7} C_VEL
LIN {X 0,Y 312.567,Z 267.052,A -85,B 0,C 180,E1 -15637.521,E2 -15637.521} C_VEL
LIN {X 0,Y 312.57,Z 267.053,A -85,B 0,C 180,E1 -15641.645,E2 -15641.645} C_VEL
LIN {X 0,Y 312.687,Z 267.038,A -85,B 0,C 180,E1 -15645.679,E2 -15645.679} C_VEL
LIN {X 0,Y 312.684,Z 267.037,A -85,B 0,C 180,E1 -15649.634,E2 -15649.634} C_VEL
LIN {X 0,Y 312.816,Z 267.017,A -85,B 0,C 180,E1 -15652.246,E2 -15652.246} C_VEL
LIN {X 0,Y 312.691,Z 267.033,A -85,B 0,C 180,E1 -15654.835,E2 -15654.835} C_VEL
LIN {X 0,Y 312.976,Z 266.997,A -85,B 0,C 180,E1 -15658.706,E2 -15658.706} C_VEL
LIN {X 0,Y 312.977,Z 266.992,A -85,B 0,C 180,E1 -15661.279,E2 -15661.279} C_VEL
LIN {X 0,Y 312.692,Z 267.035,A -85,B 0,C 180,E1 -15665.15,E2 -15665.15} C_VEL
LIN {X 0,Y 312.814,Z 267.017,A -85,B 0,C 180,E1 -15667.739,E2 -15667.739} C_VEL
LIN {X 0,Y 312.646,Z 267.038,A -85,B 0,C 180,E1 -15671.664,E2 -15671.664} C_VEL
LIN {X 0,Y 312.648,Z 267.04,A -85,B 0,C 180,E1 -15674.857,E2 -15674.857} C_VEL
LIN {X 0,Y 312.525,Z 267.053,A -85,B 0,C 180,E1 -15679.185,E2 -15679.185} C_VEL
LIN {X 0,Y 312.5,Z 267.06,A -85,B 0,C 180,E1 -15682.772,E2 -15682.772} C_VEL
LIN {X 0,Y 312.567,Z 267.047,A -85,B 0,C 180,E1 -15685.925,E2 -15685.925} C_VEL
LIN {X 0,Y 312.476,Z 267.059,A -85,B 0,C 180,E1 -15689.646,E2 -15689.646} C_VEL
LIN {X 0,Y 312.485,Z 267.058,A -85,B 0,C 180,E1 -15693.681,E2 -15693.681} C_VEL
LIN {X 0,Y 312.503,Z 267.056,A -85,B 0,C 180,E1 -15697.376,E2 -15697.376} C_VEL
LIN {X 0,Y 312.488,Z 267.059,A -85,B 0,C 180,E1 -15700.696,E2 -15700.696} C_VEL
LIN {X 0,Y 312.553,Z 267.054,A -85,B 0,C 180,E1 -15704.178,E2 -15704.178} C_VEL
LIN {X 0,Y 312.511,Z 267.058,A -85,B 0,C 180,E1 -15707.898,E2 -15707.898} C_VEL
LIN {X 0,Y 312.508,Z 267.06,A -85,B 0,C 180,E1 -15711.9,E2 -15711.9} C_VEL
LIN {X 0,Y 312.455,Z 267.067,A -85,B 0,C 180,E1 -15715.785,E2 -15715.785} C_VEL
LIN {X 0,Y 312.471,Z 267.06,A -85,B 0,C 180,E1 -15718.849,E2 -15718.849} C_VEL
LIN {X 0,Y 312.521,Z 267.058,A -85,B 0,C 180,E1 -15721.82,E2 -15721.82} C_VEL
LIN {X 0,Y 312.54,Z 267.052,A -85,B 0,C 180,E1 -15724.708,E2 -15724.708} C_VEL
LIN {X 0,Y 312.544,Z 267.053,A -85,B 0,C 180,E1 -15726.357,E2 -15726.357} C_VEL
LIN {X 0,Y 313.547,Z 269.922,A -85,B 0,C 180,E1 -15726.525,E2 -15726.525} C_VEL
LIN {X 0,Y 318.511,Z 278.002,A -85,B 0,C 180,E1 -15727.231,E2 -15727.231} C_VEL
LIN {X 0,Y 323.451,Z 284.635,A -85,B 0,C 180,E1 -15728.024,E2 -15728.024} C_VEL
LIN {X 0,Y 328.208,Z 290.515,A -85,B 0,C 180,E1 -15728.862,E2 -15728.862} C_VEL
LIN {X 0,Y 332.594,Z 295.793,A -85,B 0,C 180,E1 -15729.703,E2 -15729.703} C_VEL
LIN {X 0,Y 337.929,Z 301.838,A -85,B 0,C 180,E1 -15730.813,E2 -15730.813} C_VEL
LIN {X 0,Y 343.491,Z 307.853,A -85,B 0,C 180,E1 -15732.074,E2 -15732.074} C_VEL
LIN {X 0,Y 349.841,Z 314.343,A -85,B 0,C 180,E1 -15733.666,E2 -15733.666} C_VEL
LIN {X 0,Y 352.511,Z 316.553,A -85,B 0,C 180,E1 -15734.348,E2 -15734.348} C_VEL
LIN {X 0,Y 356.886,Z 321.133,A -85,B 0,C 180,E1 -15735.664,E2 -15735.664} C_VEL
LIN {X 0,Y 361.377,Z 325.003,A -85,B 0,C 180,E1 -15737.1,E2 -15737.1} C_VEL
LIN {X 0,Y 365.52,Z 328.901,A -85,B 0,C 180,E1 -15738.644,E2 -15738.644} C_VEL
LIN {X 0,Y 369.342,Z 331.485,A -85,B 0,C 180,E1 -15740.139,E2 -15740.139} C_VEL
LIN {X 0,Y 371.545,Z 333.846,A -85,B 0,C 180,E1 -15741.297,E2 -15741.297} C_VEL
LIN {X 0,Y 373.454,Z 335.757,A -85,B 0,C 180,E1 -15742.43,E2 -15742.43} C_VEL
LIN {X 0,Y 375.21,Z 337.191,A -85,B 0,C 180,E1 -15743.547,E2 -15743.547} C_VEL
LIN {X 0,Y 376.743,Z 338.168,A -85,B 0,C 180,E1 -15744.648,E2 -15744.648} C_VEL
LIN {X 0,Y 378.087,Z 338.723,A -85,B 0,C 180,E1 -15745.736,E2 -15745.736} C_VEL
LIN {X 0,Y 379.779,Z 339.189,A -85,B 0,C 180,E1 -15747.604,E2 -15747.604} C_VEL
LIN {X 0,Y 380.452,Z 339.309,A -85,B 0,C 180,E1 -15748.942,E2 -15748.942} C_VEL
LIN {X 0,Y 380.62,Z 339.339,A -85,B 0,C 180,E1 -15750,E2 -15750} C_VEL
LIN {X 0,Y 380.45,Z 339.313,A -85,B 0,C 180,E1 -15751.058,E2 -15751.058} C_VEL
LIN {X 0,Y 379.779,Z 339.186,A -85,B 0,C 180,E1 -15752.395,E2 -15752.395} C_VEL
LIN {X 0,Y 378.076,Z 338.759,A -85,B 0,C 180,E1 -15754.264,E2 -15754.264} C_VEL
LIN {X 0,Y 376.78,Z 338.137,A -85,B 0,C 180,E1 -15755.351,E2 -15755.351} C_VEL
LIN {X 0,Y 374.929,Z 336.979,A -85,B 0,C 180,E1 -15756.632,E2 -15756.632} C_VEL
LIN {X 0,Y 373.47,Z 335.771,A -85,B 0,C 180,E1 -15757.569,E2 -15757.569} C_VEL
LIN {X 0,Y 370.332,Z 332.493,A -85,B 0,C 180,E1 -15759.369,E2 -15759.369} C_VEL
LIN {X 0,Y 367.996,Z 330.654,A -85,B 0,C 180,E1 -15760.38,E2 -15760.38} C_VEL
LIN {X 0,Y 364.368,Z 327.982,A -85,B 0,C 180,E1 -15761.768,E2 -15761.768} C_VEL
LIN {X 0,Y 359.426,Z 323.161,A -85,B 0,C 180,E1 -15763.57,E2 -15763.57} C_VEL
LIN {X 0,Y 354.916,Z 319.295,A -85,B 0,C 180,E1 -15764.917,E2 -15764.917} C_VEL
LIN {X 0,Y 350.956,Z 315.286,A -85,B 0,C 180,E1 -15766.047,E2 -15766.047} C_VEL
LIN {X 0,Y 346.45,Z 310.893,A -85,B 0,C 180,E1 -15767.205,E2 -15767.205} C_VEL
LIN {X 0,Y 339.865,Z 304.005,A -85,B 0,C 180,E1 -15768.757,E2 -15768.757} C_VEL
LIN {X 0,Y 333.827,Z 297.242,A -85,B 0,C 180,E1 -15770.047,E2 -15770.047} C_VEL
LIN {X 0,Y 328.417,Z 290.78,A -85,B 0,C 180,E1 -15771.096,E2 -15771.096} C_VEL
LIN {X 0,Y 324.281,Z 285.677,A -85,B 0,C 180,E1 -15771.836,E2 -15771.836} C_VEL
LIN {X 0,Y 320.398,Z 280.545,A -85,B 0,C 180,E1 -15772.48,E2 -15772.48} C_VEL
LIN {X 0,Y 317.02,Z 275.63,A -85,B 0,C 180,E1 -15772.991,E2 -15772.991} C_VEL
LIN {X 0,Y 314.404,Z 271.183,A -85,B 0,C 180,E1 -15773.367,E2 -15773.367} C_VEL
LIN {X 0,Y 312.75,Z 268.112,A -85,B 0,C 180,E1 -15773.592,E2 -15773.592} C_VEL
LIN {X 0,Y 312.524,Z 267.055,A -85,B 0,C 180,E1 -15773.648,E2 -15773.648} C_VEL
LIN {X 0,Y 312.501,Z 267.059,A -85,B 0,C 180,E1 -15776.73,E2 -15776.73} C_VEL
LIN {X 0,Y 312.492,Z 267.059,A -85,B 0,C 180,E1 -15779.655,E2 -15779.655} C_VEL
LIN {X 0,Y 312.469,Z 267.062,A -85,B 0,C 180,E1 -15783.694,E2 -15783.694} C_VEL
LIN {X 0,Y 312.492,Z 267.058,A -85,B 0,C 180,E1 -15787.389,E2 -15787.389} C_VEL
LIN {X 0,Y 312.481,Z 267.059,A -85,B 0,C 180,E1 -15790.709,E2 -15790.709} C_VEL
LIN {X 0,Y 312.551,Z 267.052,A -85,B 0,C 180,E1 -15794.19,E2 -15794.19} C_VEL
LIN {X 0,Y 312.516,Z 267.059,A -85,B 0,C 180,E1 -15797.911,E2 -15797.911} C_VEL
LIN {X 0,Y 312.505,Z 267.059,A -85,B 0,C 180,E1 -15801.916,E2 -15801.916} C_VEL
LIN {X 0,Y 312.471,Z 267.063,A -85,B 0,C 180,E1 -15805.797,E2 -15805.797} C_VEL
LIN {X 0,Y 312.475,Z 267.06,A -85,B 0,C 180,E1 -15808.859,E2 -15808.859} C_VEL
LIN {X 0,Y 312.535,Z 267.054,A -85,B 0,C 180,E1 -15811.831,E2 -15811.831} C_VEL
LIN {X 0,Y 312.556,Z 267.048,A -85,B 0,C 180,E1 -15814.718,E2 -15814.718} C_VEL
LIN {X 0,Y 312.539,Z 267.055,A -85,B 0,C 180,E1 -15817.535,E2 -15817.535} C_VEL
LIN {X 0,Y 312.544,Z 267.052,A -85,B 0,C 180,E1 -15821.66,E2 -15821.66} C_VEL
LIN {X 0,Y 312.666,Z 267.035,A -85,B 0,C 180,E1 -15825.694,E2 -15825.694} C_VEL
LIN {X 0,Y 312.669,Z 267.034,A -85,B 0,C 180,E1 -15829.649,E2 -15829.649} C_VEL
LIN {X 0,Y 312.814,Z 267.017,A -85,B 0,C 180,E1 -15832.261,E2 -15832.261} C_VEL
LIN {X 0,Y 312.692,Z 267.035,A -85,B 0,C 180,E1 -15834.85,E2 -15834.85} C_VEL
LIN {X 0,Y 312.696,Z 267.027,A -85,B 0,C 180,E1 -15836.311,E2 -15836.311} C_VEL
LIN {X 0,Y 312.171,Z 267.091,A -85,B 0,C 180,E1 -15837.389,E2 -15837.389} C_VEL
LIN {X 0,Y 309.448,Z 267.433,A -85,B 0,C 180,E1 -15839.147,E2 -15839.147} C_VEL
LIN {X 0,Y 307.044,Z 267.734,A -85,B 0,C 180,E1 -15840.572,E2 -15840.572} C_VEL
LIN {X 0,Y 305.975,Z 267.868,A -85,B 0,C 180,E1 -15841.674,E2 -15841.674} C_VEL
LIN {X 0,Y 305.872,Z 267.881,A -85,B 0,C 180,E1 -15842.048,E2 -15842.048} C_VEL
LIN {X 0,Y 305.795,Z 267.896,A -85,B 0,C 180,E1 -15846.606,E2 -15846.606} C_VEL
LIN {X 0,Y 305.693,Z 267.905,A -85,B 0,C 180,E1 -15849.268,E2 -15849.268} C_VEL
LIN {X 0,Y 305.587,Z 267.918,A -85,B 0,C 180,E1 -15853.303,E2 -15853.303} C_VEL
LIN {X 0,Y 305.553,Z 267.925,A -85,B 0,C 180,E1 -15856.029,E2 -15856.029} C_VEL
LIN {X 0,Y 305.488,Z 267.934,A -85,B 0,C 180,E1 -15860.194,E2 -15860.194} C_VEL
LIN {X 0,Y 305.467,Z 267.936,A -85,B 0,C 180,E1 -15864.472,E2 -15864.472} C_VEL
LIN {X 0,Y 305.46,Z 267.935,A -85,B 0,C 180,E1 -15867.404,E2 -15867.404} C_VEL
LIN {X 0,Y 305.439,Z 267.94,A -85,B 0,C 180,E1 -15870.418,E2 -15870.418} C_VEL
LIN {X 0,Y 305.519,Z 268.134,A -85,B 0,C 180,E1 -15874.096,E2 -15874.096} C_VEL
LIN {X 0,Y 305.713,Z 269.753,A -85,B 0,C 180,E1 -15876.713,E2 -15876.713} C_VEL
LIN {X 0,Y 306.129,Z 272.465,A -85,B 0,C 180,E1 -15880.748,E2 -15880.748} C_VEL
LIN {X 0,Y 306.44,Z 275.411,A -85,B 0,C 180,E1 -15884.688,E2 -15884.688} C_VEL
LIN {X 0,Y 306.497,Z 277.466,A -85,B 0,C 180,E1 -15887.21,E2 -15887.21} C_VEL
LIN {X 0,Y 306.308,Z 279.912,A -85,B 0,C 180,E1 -15890.027,E2 -15890.027} C_VEL
LIN {X 0,Y 305.863,Z 283.146,A -85,B 0,C 180,E1 -15893.543,E2 -15893.543} C_VEL
LIN {X 0,Y 305.409,Z 285.989,A -85,B 0,C 180,E1 -15896.477,E2 -15896.477} C_VEL
LIN {X 0,Y 304.955,Z 289.065,A -85,B 0,C 180,E1 -15899.536,E2 -15899.536} C_VEL
LIN {X 0,Y 304.378,Z 293.976,A -85,B 0,C 180,E1 -15904.234,E2 -15904.234} C_VEL
LIN {X 0,Y 304.197,Z 295.868,A -85,B 0,C 180,E1 -15906.006,E2 -15906.006} C_VEL
LIN {X 0,Y 307.837,Z 310.634,A -85,B 0,C 180,E1 -15907.008,E2 -15907.008} C_VEL
LIN {X 0,Y 309.998,Z 322.71,A -85,B 0,C 180,E1 -15908.039,E2 -15908.039} C_VEL
LIN {X 0,Y 311.215,Z 332.227,A -85,B 0,C 180,E1 -15908.993,E2 -15908.993} C_VEL
LIN {X 0,Y 311.81,Z 340.197,A -85,B 0,C 180,E1 -15909.896,E2 -15909.896} C_VEL
LIN {X 0,Y 310.333,Z 350.491,A -85,B 0,C 180,E1 -15911.173,E2 -15911.173} C_VEL
LIN {X 0,Y 309.037,Z 359.02,A -85,B 0,C 180,E1 -15912.463,E2 -15912.463} C_VEL
LIN {X 0,Y 307.986,Z 366.191,A -85,B 0,C 180,E1 -15913.758,E2 -15913.758} C_VEL
LIN {X 0,Y 307.052,Z 372.444,A -85,B 0,C 180,E1 -15915.079,E2 -15915.079} C_VEL
LIN {X 0,Y 305.956,Z 378.98,A -85,B 0,C 180,E1 -15916.721,E2 -15916.721} C_VEL
LIN {X 0,Y 305.219,Z 383.481,A -85,B 0,C 180,E1 -15918.04,E2 -15918.04} C_VEL
LIN {X 0,Y 304.458,Z 388.975,A -85,B 0,C 180,E1 -15920.031,E2 -15920.031} C_VEL
LIN {X 0,Y 303.974,Z 393.302,A -85,B 0,C 180,E1 -15922.026,E2 -15922.026} C_VEL
LIN {X 0,Y 303.761,Z 395.67,A -85,B 0,C 180,E1 -15923.357,E2 -15923.357} C_VEL
LIN {X 0,Y 303.639,Z 397.471,A -85,B 0,C 180,E1 -15924.688,E2 -15924.688} C_VEL
LIN {X 0,Y 303.61,Z 399.921,A -85,B 0,C 180,E1 -15927.347,E2 -15927.347} C_VEL
LIN {X 0,Y 303.569,Z 400.51,A -85,B 0,C 180,E1 -15928.673,E2 -15928.673} C_VEL
LIN {X 0,Y 303.569,Z 400.51,A -85,B 0,C 180,E1 -15931.327,E2 -15931.327} C_VEL
LIN {X 0,Y 303.61,Z 399.921,A -85,B 0,C 180,E1 -15932.653,E2 -15932.653} C_VEL
LIN {X 0,Y 303.619,Z 397.47,A -85,B 0,C 180,E1 -15935.312,E2 -15935.312} C_VEL
LIN {X 0,Y 303.859,Z 394.52,A -85,B 0,C 180,E1 -15937.308,E2 -15937.308} C_VEL
LIN {X 0,Y 304.271,Z 390.529,A -85,B 0,C 180,E1 -15939.304,E2 -15939.304} C_VEL
LIN {X 0,Y 304.976,Z 385.399,A -85,B 0,C 180,E1 -15941.296,E2 -15941.296} C_VEL
LIN {X 0,Y 305.749,Z 380.136,A -85,B 0,C 180,E1 -15942.951,E2 -15942.951} C_VEL
LIN {X 0,Y 306.804,Z 373.82,A -85,B 0,C 180,E1 -15944.594,E2 -15944.594} C_VEL
LIN {X 0,Y 307.756,Z 367.869,A -85,B 0,C 180,E1 -15945.904,E2 -15945.904} C_VEL
LIN {X 0,Y 308.745,Z 360.94,A -85,B 0,C 180,E1 -15947.212,E2 -15947.212} C_VEL
LIN {X 0,Y 309.782,Z 353.894,A -85,B 0,C 180,E1 -15948.347,E2 -15948.347} C_VEL
LIN {X 0,Y 311.055,Z 345.603,A -85,B 0,C 180,E1 -15949.466,E2 -15949.466} C_VEL
LIN {X 0,Y 311.803,Z 338.773,A -85,B 0,C 180,E1 -15950.276,E2 -15950.276} C_VEL
LIN {X 0,Y 310.614,Z 327.103,A -85,B 0,C 180,E1 -15951.537,E2 -15951.537} C_VEL
LIN {X 0,Y 309.261,Z 317.933,A -85,B 0,C 180,E1 -15952.386,E2 -15952.386} C_VEL
LIN {X 0,Y 306.964,Z 306.92,A -85,B 0,C 180,E1 -15953.257,E2 -15953.257} C_VEL
LIN {X 0,Y 304.257,Z 296.61,A -85,B 0,C 180,E1 -15953.941,E2 -15953.941} C_VEL
LIN {X 0,Y 304.18,Z 295.877,A -85,B 0,C 180,E1 -15953.987,E2 -15953.987} C_VEL
LIN {X 0,Y 304.518,Z 292.142,A -85,B 0,C 180,E1 -15957.489,E2 -15957.489} C_VEL
LIN {X 0,Y 305.108,Z 287.966,A -85,B 0,C 180,E1 -15961.531,E2 -15961.531} C_VEL
LIN {X 0,Y 305.626,Z 284.445,A -85,B 0,C 180,E1 -15965.091,E2 -15965.091} C_VEL
LIN {X 0,Y 306.152,Z 281.047,A -85,B 0,C 180,E1 -15968.686,E2 -15968.686} C_VEL
LIN {X 0,Y 306.436,Z 278.387,A -85,B 0,C 180,E1 -15971.689,E2 -15971.689} C_VEL
LIN {X 0,Y 306.463,Z 275.411,A -85,B 0,C 180,E1 -15975.308,E2 -15975.308} C_VEL
LIN {X 0,Y 306.136,Z 272.463,A -85,B 0,C 180,E1 -15979.25,E2 -15979.25} C_VEL
LIN {X 0,Y 305.695,Z 269.572,A -85,B 0,C 180,E1 -15983.575,E2 -15983.575} C_VEL
LIN {X 0,Y 305.479,Z 267.939,A -85,B 0,C 180,E1 -15986.478,E2 -15986.478} C_VEL
LIN {X 0,Y 305.439,Z 267.941,A -85,B 0,C 180,E1 -15989.582,E2 -15989.582} C_VEL
LIN {X 0,Y 305.46,Z 267.935,A -85,B 0,C 180,E1 -15992.596,E2 -15992.596} C_VEL
LIN {X 0,Y 305.467,Z 267.936,A -85,B 0,C 180,E1 -15995.528,E2 -15995.528} C_VEL
LIN {X 0,Y 305.488,Z 267.935,A -85,B 0,C 180,E1 -15999.806,E2 -15999.806} C_VEL
LIN {X 0,Y 305.553,Z 267.924,A -85,B 0,C 180,E1 -16003.971,E2 -16003.971} C_VEL
LIN {X 0,Y 305.587,Z 267.917,A -85,B 0,C 180,E1 -16006.697,E2 -16006.697} C_VEL
LIN {X 0,Y 305.751,Z 267.9,A -85,B 0,C 180,E1 -16011.255,E2 -16011.255} C_VEL
LIN {X 0,Y 305.795,Z 267.896,A -85,B 0,C 180,E1 -16013.394,E2 -16013.394} C_VEL
LIN {X 0,Y 305.942,Z 267.873,A -85,B 0,C 180,E1 -16018.676,E2 -16018.676} C_VEL
LIN {X 0,Y 305.944,Z 267.867,A -85,B 0,C 180,E1 -16021.309,E2 -16021.309} C_VEL
LIN {X 0,Y 305.661,Z 267.912,A -85,B 0,C 180,E1 -16025.269,E2 -16025.269} C_VEL
LIN {X 0,Y 305.756,Z 267.896,A -85,B 0,C 180,E1 -16027.919,E2 -16027.919} C_VEL
LIN {X 0,Y 305.581,Z 267.918,A -85,B 0,C 180,E1 -16031.937,E2 -16031.937} C_VEL
LIN {X 0,Y 305.589,Z 267.92,A -85,B 0,C 180,E1 -16035.006,E2 -16035.006} C_VEL
LIN {X 0,Y 305.494,Z 267.932,A -85,B 0,C 180,E1 -16038.779,E2 -16038.779} C_VEL
LIN {X 0,Y 305.461,Z 267.934,A -85,B 0,C 180,E1 -16043.031,E2 -16043.031} C_VEL
LIN {X 0,Y 305.495,Z 267.93,A -85,B 0,C 180,E1 -16046.21,E2 -16046.21} C_VEL
LIN {X 0,Y 305.44,Z 267.937,A -85,B 0,C 180,E1 -16049.034,E2 -16049.034} C_VEL
LIN {X 0,Y 305.404,Z 267.941,A -85,B 0,C 180,E1 -16051.945,E2 -16051.945} C_VEL
LIN {X 0,Y 305.426,Z 267.937,A -85,B 0,C 180,E1 -16055.106,E2 -16055.106} C_VEL
LIN {X 0,Y 305.445,Z 267.938,A -85,B 0,C 180,E1 -16058.529,E2 -16058.529} C_VEL
LIN {X 0,Y 305.481,Z 267.932,A -85,B 0,C 180,E1 -16062.593,E2 -16062.593} C_VEL
LIN {X 0,Y 305.49,Z 267.932,A -85,B 0,C 180,E1 -16066.358,E2 -16066.358} C_VEL
LIN {X 0,Y 305.438,Z 267.94,A -85,B 0,C 180,E1 -16069.89,E2 -16069.89} C_VEL
LIN {X 0,Y 305.45,Z 267.938,A -85,B 0,C 180,E1 -16073.622,E2 -16073.622} C_VEL
LIN {X 0,Y 305.414,Z 267.94,A -85,B 0,C 180,E1 -16076.478,E2 -16076.478} C_VEL
LIN {X 0,Y 305.442,Z 267.937,A -85,B 0,C 180,E1 -16080.946,E2 -16080.946} C_VEL
LIN {X 0,Y 305.519,Z 267.929,A -85,B 0,C 180,E1 -16084.084,E2 -16084.084} C_VEL
LIN {X 0,Y 305.475,Z 267.936,A -85,B 0,C 180,E1 -16085.75,E2 -16085.75} C_VEL
LIN {X 0,Y 306.653,Z 271.026,A -85,B 0,C 180,E1 -16085.945,E2 -16085.945} C_VEL
LIN {X 0,Y 310.947,Z 278.724,A -85,B 0,C 180,E1 -16086.519,E2 -16086.519} C_VEL
LIN {X 0,Y 316.621,Z 287.026,A -85,B 0,C 180,E1 -16087.379,E2 -16087.379} C_VEL
LIN {X 0,Y 323.263,Z 295.316,A -85,B 0,C 180,E1 -16088.514,E2 -16088.514} C_VEL
LIN {X 0,Y 328.264,Z 301.255,A -85,B 0,C 180,E1 -16089.47,E2 -16089.47} C_VEL
LIN {X 0,Y 333.401,Z 307.167,A -85,B 0,C 180,E1 -16090.55,E2 -16090.55} C_VEL
LIN {X 0,Y 339.859,Z 314.005,A -85,B 0,C 180,E1 -16092.001,E2 -16092.001} C_VEL
LIN {X 0,Y 345.593,Z 319.886,A -85,B 0,C 180,E1 -16093.459,E2 -16093.459} C_VEL
LIN {X 0,Y 348.761,Z 322.636,A -85,B 0,C 180,E1 -16094.282,E2 -16094.282} C_VEL
LIN {X 0,Y 352.715,Z 326.785,A -85,B 0,C 180,E1 -16095.491,E2 -16095.491} C_VEL
LIN {X 0,Y 357.159,Z 330.603,A -85,B 0,C 180,E1 -16096.9,E2 -16096.9} C_VEL
LIN {X 0,Y 361.366,Z 334.616,A -85,B 0,C 180,E1 -16098.464,E2 -16098.464} C_VEL
LIN {X 0,Y 365.432,Z 337.409,A -85,B 0,C 180,E1 -16100.033,E2 -16100.033} C_VEL
LIN {X 0,Y 368.998,Z 341.077,A -85,B 0,C 180,E1 -16101.984,E2 -16101.984} C_VEL
LIN {X 0,Y 371.348,Z 343.118,A -85,B 0,C 180,E1 -16103.48,E2 -16103.48} C_VEL
LIN {X 0,Y 373.715,Z 344.507,A -85,B 0,C 180,E1 -16105.228,E2 -16105.228} C_VEL
LIN {X 0,Y 375.375,Z 345.044,A -85,B 0,C 180,E1 -16106.78,E2 -16106.78} C_VEL
LIN {X 0,Y 376.202,Z 345.251,A -85,B 0,C 180,E1 -16107.859,E2 -16107.859} C_VEL
LIN {X 0,Y 376.715,Z 345.352,A -85,B 0,C 180,E1 -16108.931,E2 -16108.931} C_VEL
LIN {X 0,Y 376.902,Z 345.37,A -85,B 0,C 180,E1 -16110,E2 -16110} C_VEL
LIN {X 0,Y 376.714,Z 345.356,A -85,B 0,C 180,E1 -16111.069,E2 -16111.069} C_VEL
LIN {X 0,Y 376.201,Z 345.244,A -85,B 0,C 180,E1 -16112.141,E2 -16112.141} C_VEL
LIN {X 0,Y 375.358,Z 345.057,A -85,B 0,C 180,E1 -16113.22,E2 -16113.22} C_VEL
LIN {X 0,Y 373.714,Z 344.498,A -85,B 0,C 180,E1 -16114.77,E2 -16114.77} C_VEL
LIN {X 0,Y 371.324,Z 343.118,A -85,B 0,C 180,E1 -16116.52,E2 -16116.52} C_VEL
LIN {X 0,Y 369.001,Z 341.07,A -85,B 0,C 180,E1 -16118.02,E2 -16118.02} C_VEL
LIN {X 0,Y 365.434,Z 337.419,A -85,B 0,C 180,E1 -16119.967,E2 -16119.967} C_VEL
LIN {X 0,Y 361.366,Z 334.586,A -85,B 0,C 180,E1 -16121.54,E2 -16121.54} C_VEL
LIN {X 0,Y 357.15,Z 330.568,A -85,B 0,C 180,E1 -16123.103,E2 -16123.103} C_VEL
LIN {X 0,Y 352.684,Z 326.745,A -85,B 0,C 180,E1 -16124.51,E2 -16124.51} C_VEL
LIN {X 0,Y 348.724,Z 322.727,A -85,B 0,C 180,E1 -16125.708,E2 -16125.708} C_VEL
LIN {X 0,Y 342.708,Z 316.97,A -85,B 0,C 180,E1 -16127.292,E2 -16127.292} C_VEL
LIN {X 0,Y 336.673,Z 310.734,A -85,B 0,C 180,E1 -16128.731,E2 -16128.731} C_VEL
LIN {X 0,Y 329.57,Z 302.834,A -85,B 0,C 180,E1 -16130.264,E2 -16130.264} C_VEL
LIN {X 0,Y 323.599,Z 295.65,A -85,B 0,C 180,E1 -16131.425,E2 -16131.425} C_VEL
LIN {X 0,Y 319.513,Z 290.653,A -85,B 0,C 180,E1 -16132.15,E2 -16132.15} C_VEL
LIN {X 0,Y 315.07,Z 284.699,A -85,B 0,C 180,E1 -16132.878,E2 -16132.878} C_VEL
LIN {X 0,Y 310.34,Z 277.816,A -85,B 0,C 180,E1 -16133.565,E2 -16133.565} C_VEL
LIN {X 0,Y 305.877,Z 269.506,A -85,B 0,C 180,E1 -16134.159,E2 -16134.159} C_VEL
LIN {X 0,Y 305.473,Z 267.936,A -85,B 0,C 180,E1 -16134.274,E2 -16134.274} C_VEL
LIN {X 0,Y 305.468,Z 267.933,A -85,B 0,C 180,E1 -16137.396,E2 -16137.396} C_VEL
LIN {X 0,Y 305.411,Z 267.943,A -85,B 0,C 180,E1 -16140.414,E2 -16140.414} C_VEL
LIN {X 0,Y 305.414,Z 267.943,A -85,B 0,C 180,E1 -16144.083,E2 -16144.083} C_VEL
LIN {X 0,Y 305.432,Z 267.938,A -85,B 0,C 180,E1 -16146.744,E2 -16146.744} C_VEL
LIN {X 0,Y 305.438,Z 267.94,A -85,B 0,C 180,E1 -16150.11,E2 -16150.11} C_VEL
LIN {X 0,Y 305.49,Z 267.932,A -85,B 0,C 180,E1 -16153.642,E2 -16153.642} C_VEL
LIN {X 0,Y 305.481,Z 267.932,A -85,B 0,C 180,E1 -16157.407,E2 -16157.407} C_VEL
LIN {X 0,Y 305.471,Z 267.936,A -85,B 0,C 180,E1 -16161.609,E2 -16161.609} C_VEL
LIN {X 0,Y 305.426,Z 267.937,A -85,B 0,C 180,E1 -16164.894,E2 -16164.894} C_VEL
LIN {X 0,Y 305.409,Z 267.939,A -85,B 0,C 180,E1 -16168.366,E2 -16168.366} C_VEL
LIN {X 0,Y 305.469,Z 267.934,A -85,B 0,C 180,E1 -16171.119,E2 -16171.119} C_VEL
LIN {X 0,Y 305.535,Z 267.923,A -85,B 0,C 180,E1 -16174.095,E2 -16174.095} C_VEL
LIN {X 0,Y 305.447,Z 267.935,A -85,B 0,C 180,E1 -16178.409,E2 -16178.409} C_VEL
LIN {X 0,Y 305.514,Z 267.927,A -85,B 0,C 180,E1 -16182.609,E2 -16182.609} C_VEL
LIN {X 0,Y 305.607,Z 267.917,A -85,B 0,C 180,E1 -16185.356,E2 -16185.356} C_VEL
LIN {X 0,Y 305.608,Z 267.915,A -85,B 0,C 180,E1 -16189.407,E2 -16189.407} C_VEL
LIN {X 0,Y 305.756,Z 267.896,A -85,B 0,C 180,E1 -16192.081,E2 -16192.081} C_VEL
LIN {X 0,Y 305.661,Z 267.912,A -85,B 0,C 180,E1 -16194.731,E2 -16194.731} C_VEL
LIN {X 0,Y 305.944,Z 267.867,A -85,B 0,C 180,E1 -16198.691,E2 -16198.691} C_VEL
LIN {X 0,Y 305.942,Z 267.873,A -85,B 0,C 180,E1 -16201.324,E2 -16201.324} C_VEL
LIN {X 0,Y 305.872,Z 267.881,A -85,B 0,C 180,E1 -16202.048,E2 -16202.048} C_VEL
LIN {X 0,Y 305.151,Z 267.975,A -85,B 0,C 180,E1 -16203.145,E2 -16203.145} C_VEL
LIN {X 0,Y 302.24,Z 268.337,A -85,B 0,C 180,E1 -16204.93,E2 -16204.93} C_VEL
LIN {X 0,Y 299.807,Z 268.641,A -85,B 0,C 180,E1 -16206.378,E2 -16206.378} C_VEL
LIN {X 0,Y 298.778,Z 268.766,A -85,B 0,C 180,E1 -16207.501,E2 -16207.501} C_VEL
LIN {X 0,Y 298.701,Z 268.776,A -85,B 0,C 180,E1 -16207.881,E2 -16207.881} C_VEL
LIN {X 0,Y 298.549,Z 268.798,A -85,B 0,C 180,E1 -16212.239,E2 -16212.239} C_VEL
LIN {X 0,Y 298.55,Z 268.795,A -85,B 0,C 180,E1 -16215.174,E2 -16215.174} C_VEL
LIN {X 0,Y 298.45,Z 268.807,A -85,B 0,C 180,E1 -16219.625,E2 -16219.625} C_VEL
LIN {X 0,Y 298.417,Z 268.812,A -85,B 0,C 180,E1 -16223.608,E2 -16223.608} C_VEL
LIN {X 0,Y 298.411,Z 268.814,A -85,B 0,C 180,E1 -16226.589,E2 -16226.589} C_VEL
LIN {X 0,Y 298.402,Z 268.816,A -85,B 0,C 180,E1 -16229.65,E2 -16229.65} C_VEL
LIN {X 0,Y 298.405,Z 268.817,A -85,B 0,C 180,E1 -16232.806,E2 -16232.806} C_VEL
LIN {X 0,Y 298.542,Z 269.5,A -85,B 0,C 180,E1 -16234.521,E2 -16234.521} C_VEL
LIN {X 0,Y 298.777,Z 271.48,A -85,B 0,C 180,E1 -16237.712,E2 -16237.712} C_VEL
LIN {X 0,Y 299.138,Z 273.85,A -85,B 0,C 180,E1 -16241.254,E2 -16241.254} C_VEL
LIN {X 0,Y 299.421,Z 276.445,A -85,B 0,C 180,E1 -16244.769,E2 -16244.769} C_VEL
LIN {X 0,Y 299.455,Z 278.315,A -85,B 0,C 180,E1 -16247.11,E2 -16247.11} C_VEL
LIN {X 0,Y 299.367,Z 279.801,A -85,B 0,C 180,E1 -16248.904,E2 -16248.904} C_VEL
LIN {X 0,Y 298.934,Z 282.814,A -85,B 0,C 180,E1 -16252.32,E2 -16252.32} C_VEL
LIN {X 0,Y 298.486,Z 285.862,A -85,B 0,C 180,E1 -16255.592,E2 -16255.592} C_VEL
LIN {X 0,Y 298.039,Z 288.942,A -85,B 0,C 180,E1 -16258.751,E2 -16258.751} C_VEL
LIN {X 0,Y 297.352,Z 293.534,A -85,B 0,C 180,E1 -16263.317,E2 -16263.317} C_VEL
LIN {X 0,Y 297.158,Z 295.695,A -85,B 0,C 180,E1 -16265.397,E2 -16265.397} C_VEL
LIN {X 0,Y 300.902,Z 310.709,A -85,B 0,C 180,E1 -16266.465,E2 -16266.465} C_VEL
LIN {X 0,Y 303.105,Z 322.662,A -85,B 0,C 180,E1 -16267.527,E2 -16267.527} C_VEL
LIN {X 0,Y 304.306,Z 332.024,A -85,B 0,C 180,E1 -16268.492,E2 -16268.492} C_VEL
LIN {X 0,Y 304.966,Z 341.354,A -85,B 0,C 180,E1 -16269.601,E2 -16269.601} C_VEL
LIN {X 0,Y 303.621,Z 350.297,A -85,B 0,C 180,E1 -16270.741,E2 -16270.741} C_VEL
LIN {X 0,Y 302.251,Z 358.825,A -85,B 0,C 180,E1 -16272.056,E2 -16272.056} C_VEL
LIN {X 0,Y 301.084,Z 366.36,A -85,B 0,C 180,E1 -16273.453,E2 -16273.453} C_VEL
LIN {X 0,Y 300.136,Z 372.248,A -85,B 0,C 180,E1 -16274.727,E2 -16274.727} C_VEL
LIN {X 0,Y 299.023,Z 378.785,A -85,B 0,C 180,E1 -16276.407,E2 -16276.407} C_VEL
LIN {X 0,Y 298.243,Z 383.286,A -85,B 0,C 180,E1 -16277.756,E2 -16277.756} C_VEL
LIN {X 0,Y 297.442,Z 388.779,A -85,B 0,C 180,E1 -16279.793,E2 -16279.793} C_VEL
LIN {X 0,Y 296.915,Z 393.107,A -85,B 0,C 180,E1 -16281.835,E2 -16281.835} C_VEL
LIN {X 0,Y 296.708,Z 395.475,A -85,B 0,C 180,E1 -16283.198,E2 -16283.198} C_VEL
LIN {X 0,Y 296.554,Z 397.276,A -85,B 0,C 180,E1 -16284.561,E2 -16284.561} C_VEL
LIN {X 0,Y 296.536,Z 399.727,A -85,B 0,C 180,E1 -16287.283,E2 -16287.283} C_VEL
LIN {X 0,Y 296.489,Z 400.315,A -85,B 0,C 180,E1 -16288.642,E2 -16288.642} C_VEL
LIN {X 0,Y 296.489,Z 400.315,A -85,B 0,C 180,E1 -16291.358,E2 -16291.358} C_VEL
LIN {X 0,Y 296.535,Z 399.727,A -85,B 0,C 180,E1 -16292.717,E2 -16292.717} C_VEL
LIN {X 0,Y 296.534,Z 397.275,A -85,B 0,C 180,E1 -16295.44,E2 -16295.44} C_VEL
LIN {X 0,Y 296.808,Z 394.325,A -85,B 0,C 180,E1 -16297.483,E2 -16297.483} C_VEL
LIN {X 0,Y 297.245,Z 390.334,A -85,B 0,C 180,E1 -16299.526,E2 -16299.526} C_VEL
LIN {X 0,Y 297.968,Z 385.203,A -85,B 0,C 180,E1 -16301.565,E2 -16301.565} C_VEL
LIN {X 0,Y 298.814,Z 379.94,A -85,B 0,C 180,E1 -16303.256,E2 -16303.256} C_VEL
LIN {X 0,Y 299.895,Z 373.624,A -85,B 0,C 180,E1 -16304.938,E2 -16304.938} C_VEL
LIN {X 0,Y 300.923,Z 367.674,A -85,B 0,C 180,E1 -16306.275,E2 -16306.275} C_VEL
LIN {X 0,Y 301.941,Z 360.744,A -85,B 0,C 180,E1 -16307.613,E2 -16307.613} C_VEL
LIN {X 0,Y 303.204,Z 352.564,A -85,B 0,C 180,E1 -16308.935,E2 -16308.935} C_VEL
LIN {X 0,Y 304.549,Z 344.056,A -85,B 0,C 180,E1 -16310.076,E2 -16310.076} C_VEL
LIN {X 0,Y 304.986,Z 339.997,A -85,B 0,C 180,E1 -16310.573,E2 -16310.573} C_VEL
LIN {X 0,Y 303.975,Z 328.861,A -85,B 0,C 180,E1 -16311.859,E2 -16311.859} C_VEL
LIN {X 0,Y 302.377,Z 317.841,A -85,B 0,C 180,E1 -16312.917,E2 -16312.917} C_VEL
LIN {X 0,Y 299.926,Z 306.623,A -85,B 0,C 180,E1 -16313.84,E2 -16313.84} C_VEL
LIN {X 0,Y 297.22,Z 296.416,A -85,B 0,C 180,E1 -16314.545,E2 -16314.545} C_VEL
LIN {X 0,Y 297.155,Z 295.699,A -85,B 0,C 180,E1 -16314.6,E2 -16314.6} C_VEL
LIN {X 0,Y 297.657,Z 291.044,A -85,B 0,C 180,E1 -16319.109,E2 -16319.109} C_VEL
LIN {X 0,Y 298.196,Z 287.352,A -85,B 0,C 180,E1 -16322.824,E2 -16322.824} C_VEL
LIN {X 0,Y 298.702,Z 284.316,A -85,B 0,C 180,E1 -16326.029,E2 -16326.029} C_VEL
LIN {X 0,Y 299.174,Z 281.276,A -85,B 0,C 180,E1 -16329.364,E2 -16329.364} C_VEL
LIN {X 0,Y 299.437,Z 278.288,A -85,B 0,C 180,E1 -16332.893,E2 -16332.893} C_VEL
LIN {X 0,Y 299.439,Z 276.423,A -85,B 0,C 180,E1 -16335.234,E2 -16335.234} C_VEL
LIN {X 0,Y 299.146,Z 273.762,A -85,B 0,C 180,E1 -16338.859,E2 -16338.859} C_VEL
LIN {X 0,Y 298.777,Z 271.457,A -85,B 0,C 180,E1 -16342.289,E2 -16342.289} C_VEL
LIN {X 0,Y 298.52,Z 269.44,A -85,B 0,C 180,E1 -16345.589,E2 -16345.589} C_VEL
LIN {X 0,Y 298.405,Z 268.82,A -85,B 0,C 180,E1 -16347.194,E2 -16347.194} C_VEL
LIN {X 0,Y 298.411,Z 268.814,A -85,B 0,C 180,E1 -16350.619,E2 -16350.619} C_VEL
LIN {X 0,Y 298.432,Z 268.81,A -85,B 0,C 180,E1 -16354.912,E2 -16354.912} C_VEL
LIN {X 0,Y 298.412,Z 268.817,A -85,B 0,C 180,E1 -16357.856,E2 -16357.856} C_VEL
LIN {X 0,Y 298.468,Z 268.805,A -85,B 0,C 180,E1 -16360.745,E2 -16360.745} C_VEL
LIN {X 0,Y 298.589,Z 268.79,A -85,B 0,C 180,E1 -16364.987,E2 -16364.987} C_VEL
LIN {X 0,Y 298.582,Z 268.792,A -85,B 0,C 180,E1 -16369.139,E2 -16369.139} C_VEL
LIN {X 0,Y 298.707,Z 268.776,A -85,B 0,C 180,E1 -16371.877,E2 -16371.877} C_VEL
LIN {X 0,Y 298.631,Z 268.784,A -85,B 0,C 180,E1 -16374.591,E2 -16374.591} C_VEL
LIN {X 0,Y 298.909,Z 268.749,A -85,B 0,C 180,E1 -16378.645,E2 -16378.645} C_VEL
LIN {X 0,Y 298.911,Z 268.741,A -85,B 0,C 180,E1 -16381.339,E2 -16381.339} C_VEL
LIN {X 0,Y 298.631,Z 268.786,A -85,B 0,C 180,E1 -16385.393,E2 -16385.393} C_VEL
LIN {X 0,Y 298.702,Z 268.774,A -85,B 0,C 180,E1 -16388.107,E2 -16388.107} C_VEL
LIN {X 0,Y 298.532,Z 268.797,A -85,B 0,C 180,E1 -16392.224,E2 -16392.224} C_VEL
LIN {X 0,Y 298.529,Z 268.798,A -85,B 0,C 180,E1 -16395.159,E2 -16395.159} C_VEL
LIN {X 0,Y 298.422,Z 268.807,A -85,B 0,C 180,E1 -16399.61,E2 -16399.61} C_VEL
LIN {X 0,Y 298.403,Z 268.811,A -85,B 0,C 180,E1 -16403.592,E2 -16403.592} C_VEL
LIN {X 0,Y 298.455,Z 268.81,A -85,B 0,C 180,E1 -16406.567,E2 -16406.567} C_VEL
LIN {X 0,Y 298.373,Z 268.816,A -85,B 0,C 180,E1 -16409.635,E2 -16409.635} C_VEL
LIN {X 0,Y 298.359,Z 268.819,A -85,B 0,C 180,E1 -16412.793,E2 -16412.793} C_VEL
LIN {X 0,Y 298.429,Z 268.811,A -85,B 0,C 180,E1 -16416.805,E2 -16416.805} C_VEL
LIN {X 0,Y 298.415,Z 268.811,A -85,B 0,C 180,E1 -16421.243,E2 -16421.243} C_VEL
LIN {X 0,Y 298.447,Z 268.806,A -85,B 0,C 180,E1 -16425.054,E2 -16425.054} C_VEL
LIN {X 0,Y 298.408,Z 268.812,A -85,B 0,C 180,E1 -16428.892,E2 -16428.892} C_VEL
LIN {X 0,Y 298.404,Z 268.813,A -85,B 0,C 180,E1 -16433.186,E2 -16433.186} C_VEL
LIN {X 0,Y 298.345,Z 268.821,A -85,B 0,C 180,E1 -16437.194,E2 -16437.194} C_VEL
LIN {X 0,Y 298.379,Z 268.816,A -85,B 0,C 180,E1 -16440.61,E2 -16440.61} C_VEL
LIN {X 0,Y 298.431,Z 268.813,A -85,B 0,C 180,E1 -16443.47,E2 -16443.47} C_VEL
LIN {X 0,Y 298.442,Z 268.812,A -85,B 0,C 180,E1 -16445.175,E2 -16445.175} C_VEL
LIN {X 0,Y 299.444,Z 271.662,A -85,B 0,C 180,E1 -16445.339,E2 -16445.339} C_VEL
LIN {X 0,Y 304.44,Z 281.326,A -85,B 0,C 180,E1 -16446.058,E2 -16446.058} C_VEL
LIN {X 0,Y 309.571,Z 288.953,A -85,B 0,C 180,E1 -16446.818,E2 -16446.818} C_VEL
LIN {X 0,Y 315.088,Z 296.335,A -85,B 0,C 180,E1 -16447.718,E2 -16447.718} C_VEL
LIN {X 0,Y 321.701,Z 304.49,A -85,B 0,C 180,E1 -16448.941,E2 -16448.941} C_VEL
LIN {X 0,Y 328.375,Z 312.023,A -85,B 0,C 180,E1 -16450.309,E2 -16450.309} C_VEL
LIN {X 0,Y 334.186,Z 318.295,A -85,B 0,C 180,E1 -16451.612,E2 -16451.612} C_VEL
LIN {X 0,Y 340.54,Z 324.82,A -85,B 0,C 180,E1 -16453.207,E2 -16453.207} C_VEL
LIN {X 0,Y 344.987,Z 328.953,A -85,B 0,C 180,E1 -16454.397,E2 -16454.397} C_VEL
LIN {X 0,Y 348.444,Z 332.452,A -85,B 0,C 180,E1 -16455.459,E2 -16455.459} C_VEL
LIN {X 0,Y 353.32,Z 336.722,A -85,B 0,C 180,E1 -16457.032,E2 -16457.032} C_VEL
LIN {X 0,Y 357.714,Z 340.741,A -85,B 0,C 180,E1 -16458.67,E2 -16458.67} C_VEL
LIN {X 0,Y 360.943,Z 342.945,A -85,B 0,C 180,E1 -16459.908,E2 -16459.908} C_VEL
LIN {X 0,Y 363.206,Z 345.246,A -85,B 0,C 180,E1 -16461.095,E2 -16461.095} C_VEL
LIN {X 0,Y 365.178,Z 347.178,A -85,B 0,C 180,E1 -16462.258,E2 -16462.258} C_VEL
LIN {X 0,Y 367.525,Z 349.092,A -85,B 0,C 180,E1 -16463.824,E2 -16463.824} C_VEL
LIN {X 0,Y 369.917,Z 350.349,A -85,B 0,C 180,E1 -16465.642,E2 -16465.642} C_VEL
LIN {X 0,Y 371.104,Z 350.731,A -85,B 0,C 180,E1 -16466.743,E2 -16466.743} C_VEL
LIN {X 0,Y 371.974,Z 350.972,A -85,B 0,C 180,E1 -16467.834,E2 -16467.834} C_VEL
LIN {X 0,Y 372.527,Z 351.082,A -85,B 0,C 180,E1 -16468.919,E2 -16468.919} C_VEL
LIN {X 0,Y 372.722,Z 351.11,A -85,B 0,C 180,E1 -16470,E2 -16470} C_VEL
LIN {X 0,Y 372.493,Z 351.086,A -85,B 0,C 180,E1 -16471.136,E2 -16471.136} C_VEL
LIN {X 0,Y 371.972,Z 350.968,A -85,B 0,C 180,E1 -16472.166,E2 -16472.166} C_VEL
LIN {X 0,Y 371.077,Z 350.755,A -85,B 0,C 180,E1 -16473.257,E2 -16473.257} C_VEL
LIN {X 0,Y 369.914,Z 350.356,A -85,B 0,C 180,E1 -16474.358,E2 -16474.358} C_VEL
LIN {X 0,Y 367.531,Z 349.076,A -85,B 0,C 180,E1 -16476.184,E2 -16476.184} C_VEL
LIN {X 0,Y 365.177,Z 347.171,A -85,B 0,C 180,E1 -16477.742,E2 -16477.742} C_VEL
LIN {X 0,Y 362.923,Z 344.846,A -85,B 0,C 180,E1 -16479.091,E2 -16479.091} C_VEL
LIN {X 0,Y 360.943,Z 342.929,A -85,B 0,C 180,E1 -16480.092,E2 -16480.092} C_VEL
LIN {X 0,Y 356.206,Z 339.488,A -85,B 0,C 180,E1 -16481.896,E2 -16481.896} C_VEL
LIN {X 0,Y 351.845,Z 335.276,A -85,B 0,C 180,E1 -16483.491,E2 -16483.491} C_VEL
LIN {X 0,Y 345.981,Z 330.045,A -85,B 0,C 180,E1 -16485.311,E2 -16485.311} C_VEL
LIN {X 0,Y 339.569,Z 323.809,A -85,B 0,C 180,E1 -16487.055,E2 -16487.055} C_VEL
LIN {X 0,Y 331.998,Z 315.956,A -85,B 0,C 180,E1 -16488.897,E2 -16488.897} C_VEL
LIN {X 0,Y 326.123,Z 309.556,A -85,B 0,C 180,E1 -16490.169,E2 -16490.169} C_VEL
LIN {X 0,Y 319.425,Z 301.659,A -85,B 0,C 180,E1 -16491.506,E2 -16491.506} C_VEL
LIN {X 0,Y 311.838,Z 292.205,A -85,B 0,C 180,E1 -16492.82,E2 -16492.82} C_VEL
LIN {X 0,Y 306.427,Z 284.331,A -85,B 0,C 180,E1 -16493.652,E2 -16493.652} C_VEL
LIN {X 0,Y 301.717,Z 276.388,A -85,B 0,C 180,E1 -16494.333,E2 -16494.333} C_VEL
LIN {X 0,Y 298.626,Z 269.774,A -85,B 0,C 180,E1 -16494.783,E2 -16494.783} C_VEL
LIN {X 0,Y 298.433,Z 268.812,A -85,B 0,C 180,E1 -16494.85,E2 -16494.85} C_VEL
LIN {X 0,Y 298.41,Z 268.815,A -85,B 0,C 180,E1 -16498.1,E2 -16498.1} C_VEL
LIN {X 0,Y 298.344,Z 268.824,A -85,B 0,C 180,E1 -16502.021,E2 -16502.021} C_VEL
LIN {X 0,Y 298.383,Z 268.819,A -85,B 0,C 180,E1 -16506.074,E2 -16506.074} C_VEL
LIN {X 0,Y 298.383,Z 268.816,A -85,B 0,C 180,E1 -16509.489,E2 -16509.489} C_VEL
LIN {X 0,Y 298.426,Z 268.809,A -85,B 0,C 180,E1 -16513.124,E2 -16513.124} C_VEL
LIN {X 0,Y 298.429,Z 268.809,A -85,B 0,C 180,E1 -16516.94,E2 -16516.94} C_VEL
LIN {X 0,Y 298.392,Z 268.814,A -85,B 0,C 180,E1 -16521.007,E2 -16521.007} C_VEL
LIN {X 0,Y 298.395,Z 268.816,A -85,B 0,C 180,E1 -16523.939,E2 -16523.939} C_VEL
LIN {X 0,Y 298.356,Z 268.82,A -85,B 0,C 180,E1 -16527.993,E2 -16527.993} C_VEL
LIN {X 0,Y 298.411,Z 268.813,A -85,B 0,C 180,E1 -16531.91,E2 -16531.91} C_VEL
LIN {X 0,Y 298.453,Z 268.806,A -85,B 0,C 180,E1 -16534.931,E2 -16534.931} C_VEL
LIN {X 0,Y 298.397,Z 268.815,A -85,B 0,C 180,E1 -16539.321,E2 -16539.321} C_VEL
LIN {X 0,Y 298.444,Z 268.807,A -85,B 0,C 180,E1 -16542.183,E2 -16542.183} C_VEL
LIN {X 0,Y 298.567,Z 268.794,A -85,B 0,C 180,E1 -16545.003,E2 -16545.003} C_VEL
LIN {X 0,Y 298.567,Z 268.794,A -85,B 0,C 180,E1 -16549.154,E2 -16549.154} C_VEL
LIN {X 0,Y 298.702,Z 268.774,A -85,B 0,C 180,E1 -16551.893,E2 -16551.893} C_VEL
LIN {X 0,Y 298.631,Z 268.786,A -85,B 0,C 180,E1 -16554.607,E2 -16554.607} C_VEL
LIN {X 0,Y 298.911,Z 268.741,A -85,B 0,C 180,E1 -16558.661,E2 -16558.661} C_VEL
LIN {X 0,Y 298.909,Z 268.749,A -85,B 0,C 180,E1 -16561.355,E2 -16561.355} C_VEL
LIN {X 0,Y 298.743,Z 268.774,A -85,B 0,C 180,E1 -16566.763,E2 -16566.763} C_VEL
LIN {X 0,Y 298.701,Z 268.776,A -85,B 0,C 180,E1 -16567.881,E2 -16567.881} C_VEL
LIN {X 0,Y 298.026,Z 268.864,A -85,B 0,C 180,E1 -16569.005,E2 -16569.005} C_VEL
LIN {X 0,Y 295.085,Z 269.229,A -85,B 0,C 180,E1 -16570.833,E2 -16570.833} C_VEL
LIN {X 0,Y 292.606,Z 269.539,A -85,B 0,C 180,E1 -16572.316,E2 -16572.316} C_VEL
LIN {X 0,Y 291.576,Z 269.664,A -85,B 0,C 180,E1 -16573.468,E2 -16573.468} C_VEL
LIN {X 0,Y 291.511,Z 269.673,A -85,B 0,C 180,E1 -16573.858,E2 -16573.858} C_VEL
LIN {X 0,Y 291.431,Z 269.683,A -85,B 0,C 180,E1 -16576.829,E2 -16576.829} C_VEL
LIN {X 0,Y 291.397,Z 269.687,A -85,B 0,C 180,E1 -16579.849,E2 -16579.849} C_VEL
LIN {X 0,Y 291.355,Z 269.695,A -85,B 0,C 180,E1 -16584.216,E2 -16584.216} C_VEL
LIN {X 0,Y 291.359,Z 269.691,A -85,B 0,C 180,E1 -16587.285,E2 -16587.285} C_VEL
LIN {X 0,Y 291.328,Z 269.698,A -85,B 0,C 180,E1 -16590.445,E2 -16590.445} C_VEL
LIN {X 0,Y 291.35,Z 269.698,A -85,B 0,C 180,E1 -16592.408,E2 -16592.408} C_VEL
LIN {X 0,Y 291.56,Z 271.097,A -85,B 0,C 180,E1 -16595.354,E2 -16595.354} C_VEL
LIN {X 0,Y 291.941,Z 273.771,A -85,B 0,C 180,E1 -16599.617,E2 -16599.617} C_VEL
LIN {X 0,Y 292.19,Z 275.626,A -85,B 0,C 180,E1 -16602.344,E2 -16602.344} C_VEL
LIN {X 0,Y 292.388,Z 278.201,A -85,B 0,C 180,E1 -16605.81,E2 -16605.81} C_VEL
LIN {X 0,Y 292.343,Z 280.087,A -85,B 0,C 180,E1 -16608.188,E2 -16608.188} C_VEL
LIN {X 0,Y 292.034,Z 282.696,A -85,B 0,C 180,E1 -16611.267,E2 -16611.267} C_VEL
LIN {X 0,Y 291.484,Z 286.124,A -85,B 0,C 180,E1 -16615.072,E2 -16615.072} C_VEL
LIN {X 0,Y 291.07,Z 288.797,A -85,B 0,C 180,E1 -16617.914,E2 -16617.914} C_VEL
LIN {X 0,Y 290.566,Z 291.846,A -85,B 0,C 180,E1 -16621.07,E2 -16621.07} C_VEL
LIN {X 0,Y 290.151,Z 295.654,A -85,B 0,C 180,E1 -16624.797,E2 -16624.797} C_VEL
LIN {X 0,Y 291.568,Z 301.067,A -85,B 0,C 180,E1 -16625.144,E2 -16625.144} C_VEL
LIN {X 0,Y 294.361,Z 312.517,A -85,B 0,C 180,E1 -16626.054,E2 -16626.054} C_VEL
LIN {X 0,Y 296.382,Z 323.329,A -85,B 0,C 180,E1 -16627.067,E2 -16627.067} C_VEL
LIN {X 0,Y 297.512,Z 332.773,A -85,B 0,C 180,E1 -16628.082,E2 -16628.082} C_VEL
LIN {X 0,Y 298.181,Z 341.205,A -85,B 0,C 180,E1 -16629.122,E2 -16629.122} C_VEL
LIN {X 0,Y 296.917,Z 350.102,A -85,B 0,C 180,E1 -16630.288,E2 -16630.288} C_VEL
LIN {X 0,Y 295.467,Z 358.629,A -85,B 0,C 180,E1 -16631.63,E2 -16631.63} C_VEL
LIN {X 0,Y 294.372,Z 365.562,A -85,B 0,C 180,E1 -16632.932,E2 -16632.932} C_VEL
LIN {X 0,Y 293.234,Z 372.052,A -85,B 0,C 180,E1 -16634.358,E2 -16634.358} C_VEL
LIN {X 0,Y 292.093,Z 378.59,A -85,B 0,C 180,E1 -16636.078,E2 -16636.078} C_VEL
LIN {X 0,Y 291.275,Z 383.09,A -85,B 0,C 180,E1 -16637.458,E2 -16637.458} C_VEL
LIN {X 0,Y 290.442,Z 388.584,A -85,B 0,C 180,E1 -16639.544,E2 -16639.544} C_VEL
LIN {X 0,Y 289.873,Z 392.911,A -85,B 0,C 180,E1 -16641.636,E2 -16641.636} C_VEL
LIN {X 0,Y 289.627,Z 395.28,A -85,B 0,C 180,E1 -16643.031,E2 -16643.031} C_VEL
LIN {X 0,Y 289.449,Z 397.323,A -85,B 0,C 180,E1 -16644.615,E2 -16644.615} C_VEL
LIN {X 0,Y 289.439,Z 399.532,A -85,B 0,C 180,E1 -16647.217,E2 -16647.217} C_VEL
LIN {X 0,Y 289.412,Z 400.121,A -85,B 0,C 180,E1 -16648.609,E2 -16648.609} C_VEL
LIN {X 0,Y 289.412,Z 400.121,A -85,B 0,C 180,E1 -16651.391,E2 -16651.391} C_VEL
LIN {X 0,Y 289.439,Z 399.532,A -85,B 0,C 180,E1 -16652.783,E2 -16652.783} C_VEL
LIN {X 0,Y 289.458,Z 397.08,A -85,B 0,C 180,E1 -16655.573,E2 -16655.573} C_VEL
LIN {X 0,Y 289.739,Z 394.129,A -85,B 0,C 180,E1 -16657.666,E2 -16657.666} C_VEL
LIN {X 0,Y 290.202,Z 390.138,A -85,B 0,C 180,E1 -16659.76,E2 -16659.76} C_VEL
LIN {X 0,Y 290.979,Z 385.007,A -85,B 0,C 180,E1 -16661.847,E2 -16661.847} C_VEL
LIN {X 0,Y 291.89,Z 379.745,A -85,B 0,C 180,E1 -16663.577,E2 -16663.577} C_VEL
LIN {X 0,Y 292.993,Z 373.428,A -85,B 0,C 180,E1 -16665.299,E2 -16665.299} C_VEL
LIN {X 0,Y 294.264,Z 366.479,A -85,B 0,C 180,E1 -16666.874,E2 -16666.874} C_VEL
LIN {X 0,Y 295.413,Z 358.628,A -85,B 0,C 180,E1 -16668.374,E2 -16668.374} C_VEL
LIN {X 0,Y 296.887,Z 350.101,A -85,B 0,C 180,E1 -16669.714,E2 -16669.714} C_VEL
LIN {X 0,Y 298.175,Z 341.208,A -85,B 0,C 180,E1 -16670.878,E2 -16670.878} C_VEL
LIN {X 0,Y 297.257,Z 330.175,A -85,B 0,C 180,E1 -16672.227,E2 -16672.227} C_VEL
LIN {X 0,Y 295.48,Z 317.864,A -85,B 0,C 180,E1 -16673.467,E2 -16673.467} C_VEL
LIN {X 0,Y 292.97,Z 306.5,A -85,B 0,C 180,E1 -16674.438,E2 -16674.438} C_VEL
LIN {X 0,Y 290.241,Z 296.452,A -85,B 0,C 180,E1 -16675.167,E2 -16675.167} C_VEL
LIN {X 0,Y 290.149,Z 295.524,A -85,B 0,C 180,E1 -16675.239,E2 -16675.239} C_VEL
LIN {X 0,Y 290.644,Z 291.268,A -85,B 0,C 180,E1 -16679.472,E2 -16679.472} C_VEL
LIN {X 0,Y 291.278,Z 287.198,A -85,B 0,C 180,E1 -16683.706,E2 -16683.706} C_VEL
LIN {X 0,Y 291.854,Z 283.867,A -85,B 0,C 180,E1 -16687.368,E2 -16687.368} C_VEL
LIN {X 0,Y 292.23,Z 281.166,A -85,B 0,C 180,E1 -16690.49,E2 -16690.49} C_VEL
LIN {X 0,Y 292.392,Z 278.45,A -85,B 0,C 180,E1 -16693.848,E2 -16693.848} C_VEL
LIN {X 0,Y 292.323,Z 276.702,A -85,B 0,C 180,E1 -16696.157,E2 -16696.157} C_VEL
LIN {X 0,Y 292.043,Z 274.363,A -85,B 0,C 180,E1 -16699.469,E2 -16699.469} C_VEL
LIN {X 0,Y 291.692,Z 272.111,A -85,B 0,C 180,E1 -16702.954,E2 -16702.954} C_VEL
LIN {X 0,Y 291.428,Z 270.144,A -85,B 0,C 180,E1 -16706.305,E2 -16706.305} C_VEL
LIN {X 0,Y 291.376,Z 269.696,A -85,B 0,C 180,E1 -16707.944,E2 -16707.944} C_VEL
LIN {X 0,Y 291.352,Z 269.693,A -85,B 0,C 180,E1 -16711.148,E2 -16711.148} C_VEL
LIN {X 0,Y 291.357,Z 269.693,A -85,B 0,C 180,E1 -16714.259,E2 -16714.259} C_VEL
LIN {X 0,Y 291.368,Z 269.692,A -85,B 0,C 180,E1 -16717.291,E2 -16717.291} C_VEL
LIN {X 0,Y 291.397,Z 269.687,A -85,B 0,C 180,E1 -16720.259,E2 -16720.259} C_VEL
LIN {X 0,Y 291.501,Z 269.672,A -85,B 0,C 180,E1 -16724.658,E2 -16724.658} C_VEL
LIN {X 0,Y 291.528,Z 269.67,A -85,B 0,C 180,E1 -16728.873,E2 -16728.873} C_VEL
LIN {X 0,Y 291.659,Z 269.656,A -85,B 0,C 180,E1 -16731.679,E2 -16731.679} C_VEL
LIN {X 0,Y 291.601,Z 269.66,A -85,B 0,C 180,E1 -16734.46,E2 -16734.46} C_VEL
LIN {X 0,Y 291.875,Z 269.625,A -85,B 0,C 180,E1 -16738.612,E2 -16738.612} C_VEL
LIN {X 0,Y 291.877,Z 269.616,A -85,B 0,C 180,E1 -16741.372,E2 -16741.372} C_VEL
LIN {X 0,Y 291.691,Z 269.652,A -85,B 0,C 180,E1 -16746.911,E2 -16746.911} C_VEL
LIN {X 0,Y 291.553,Z 269.664,A -85,B 0,C 180,E1 -16749.706,E2 -16749.706} C_VEL
LIN {X 0,Y 291.496,Z 269.671,A -85,B 0,C 180,E1 -16753.942,E2 -16753.942} C_VEL
LIN {X 0,Y 291.408,Z 269.688,A -85,B 0,C 180,E1 -16756.813,E2 -16756.813} C_VEL
LIN {X 0,Y 291.369,Z 269.685,A -85,B 0,C 180,E1 -16759.834,E2 -16759.834} C_VEL
LIN {X 0,Y 291.355,Z 269.691,A -85,B 0,C 180,E1 -16764.199,E2 -16764.199} C_VEL
LIN {X 0,Y 291.383,Z 269.687,A -85,B 0,C 180,E1 -16767.265,E2 -16767.265} C_VEL
LIN {X 0,Y 291.292,Z 269.702,A -85,B 0,C 180,E1 -16770.431,E2 -16770.431} C_VEL
LIN {X 0,Y 291.31,Z 269.696,A -85,B 0,C 180,E1 -16773.691,E2 -16773.691} C_VEL
LIN {X 0,Y 291.361,Z 269.69,A -85,B 0,C 180,E1 -16777.252,E2 -16777.252} C_VEL
LIN {X 0,Y 291.363,Z 269.691,A -85,B 0,C 180,E1 -16780.624,E2 -16780.624} C_VEL
LIN {X 0,Y 291.365,Z 269.691,A -85,B 0,C 180,E1 -16784.373,E2 -16784.373} C_VEL
LIN {X 0,Y 291.344,Z 269.694,A -85,B 0,C 180,E1 -16788.384,E2 -16788.384} C_VEL
LIN {X 0,Y 291.336,Z 269.693,A -85,B 0,C 180,E1 -16791.157,E2 -16791.157} C_VEL
LIN {X 0,Y 291.337,Z 269.694,A -85,B 0,C 180,E1 -16794.624,E2 -16794.624} C_VEL
LIN {X 0,Y 291.321,Z 269.699,A -85,B 0,C 180,E1 -16797.945,E2 -16797.945} C_VEL
LIN {X 0,Y 291.33,Z 269.696,A -85,B 0,C 180,E1 -16801.153,E2 -16801.153} C_VEL
LIN {X 0,Y 291.4,Z 269.687,A -85,B 0,C 180,E1 -16804.528,E2 -16804.528} C_VEL
LIN {X 0,Y 292.553,Z 272.787,A -85,B 0,C 180,E1 -16804.742,E2 -16804.742} C_VEL
LIN {X 0,Y 297.704,Z 283.19,A -85,B 0,C 180,E1 -16805.551,E2 -16805.551} C_VEL
LIN {X 0,Y 302.875,Z 291.656,A -85,B 0,C 180,E1 -16806.402,E2 -16806.402} C_VEL
LIN {X 0,Y 309.656,Z 300.796,A -85,B 0,C 180,E1 -16807.535,E2 -16807.535} C_VEL
LIN {X 0,Y 316.53,Z 309.294,A -85,B 0,C 180,E1 -16808.804,E2 -16808.804} C_VEL
LIN {X 0,Y 322.9,Z 316.536,A -85,B 0,C 180,E1 -16810.105,E2 -16810.105} C_VEL
LIN {X 0,Y 329.54,Z 323.664,A -85,B 0,C 180,E1 -16811.594,E2 -16811.594} C_VEL
LIN {X 0,Y 335.819,Z 330.122,A -85,B 0,C 180,E1 -16813.19,E2 -16813.19} C_VEL
LIN {X 0,Y 340.463,Z 334.46,A -85,B 0,C 180,E1 -16814.434,E2 -16814.434} C_VEL
LIN {X 0,Y 345.091,Z 338.904,A -85,B 0,C 180,E1 -16815.855,E2 -16815.855} C_VEL
LIN {X 0,Y 350.117,Z 343.548,A -85,B 0,C 180,E1 -16817.574,E2 -16817.574} C_VEL
LIN {X 0,Y 354.298,Z 346.973,A -85,B 0,C 180,E1 -16819.149,E2 -16819.149} C_VEL
LIN {X 0,Y 356.643,Z 348.635,A -85,B 0,C 180,E1 -16820.105,E2 -16820.105} C_VEL
LIN {X 0,Y 360.252,Z 352.287,A -85,B 0,C 180,E1 -16822.151,E2 -16822.151} C_VEL
LIN {X 0,Y 362.065,Z 353.808,A -85,B 0,C 180,E1 -16823.312,E2 -16823.312} C_VEL
LIN {X 0,Y 363.656,Z 354.928,A -85,B 0,C 180,E1 -16824.455,E2 -16824.455} C_VEL
LIN {X 0,Y 366.099,Z 356.003,A -85,B 0,C 180,E1 -16826.439,E2 -16826.439} C_VEL
LIN {X 0,Y 367.306,Z 356.351,A -85,B 0,C 180,E1 -16827.807,E2 -16827.807} C_VEL
LIN {X 0,Y 367.893,Z 356.486,A -85,B 0,C 180,E1 -16828.905,E2 -16828.905} C_VEL
LIN {X 0,Y 368.112,Z 356.511,A -85,B 0,C 180,E1 -16830,E2 -16830} C_VEL
LIN {X 0,Y 367.893,Z 356.487,A -85,B 0,C 180,E1 -16831.095,E2 -16831.095} C_VEL
LIN {X 0,Y 367.302,Z 356.351,A -85,B 0,C 180,E1 -16832.193,E2 -16832.193} C_VEL
LIN {X 0,Y 366.094,Z 356.019,A -85,B 0,C 180,E1 -16833.549,E2 -16833.549} C_VEL
LIN {X 0,Y 363.707,Z 354.899,A -85,B 0,C 180,E1 -16835.544,E2 -16835.544} C_VEL
LIN {X 0,Y 361.238,Z 353.145,A -85,B 0,C 180,E1 -16837.231,E2 -16837.231} C_VEL
LIN {X 0,Y 358.31,Z 350.28,A -85,B 0,C 180,E1 -16839.028,E2 -16839.028} C_VEL
LIN {X 0,Y 355.875,Z 348.032,A -85,B 0,C 180,E1 -16840.238,E2 -16840.238} C_VEL
LIN {X 0,Y 351.757,Z 345.022,A -85,B 0,C 180,E1 -16841.811,E2 -16841.811} C_VEL
LIN {X 0,Y 346.956,Z 340.426,A -85,B 0,C 180,E1 -16843.562,E2 -16843.562} C_VEL
LIN {X 0,Y 342.04,Z 336.098,A -85,B 0,C 180,E1 -16845.085,E2 -16845.085} C_VEL
LIN {X 0,Y 337.108,Z 331.255,A -85,B 0,C 180,E1 -16846.5,E2 -16846.5} C_VEL
LIN {X 0,Y 330.743,Z 324.819,A -85,B 0,C 180,E1 -16848.123,E2 -16848.123} C_VEL
LIN {X 0,Y 324.766,Z 318.451,A -85,B 0,C 180,E1 -16849.507,E2 -16849.507} C_VEL
LIN {X 0,Y 318.068,Z 310.937,A -85,B 0,C 180,E1 -16850.912,E2 -16850.912} C_VEL
LIN {X 0,Y 311.143,Z 302.738,A -85,B 0,C 180,E1 -16852.195,E2 -16852.195} C_VEL
LIN {X 0,Y 304.615,Z 294.055,A -85,B 0,C 180,E1 -16853.314,E2 -16853.314} C_VEL
LIN {X 0,Y 298.804,Z 285.249,A -85,B 0,C 180,E1 -16854.266,E2 -16854.266} C_VEL
LIN {X 0,Y 294.159,Z 276.215,A -85,B 0,C 180,E1 -16855.013,E2 -16855.013} C_VEL
LIN {X 0,Y 291.576,Z 270.597,A -85,B 0,C 180,E1 -16855.408,E2 -16855.408} C_VEL
LIN {X 0,Y 291.389,Z 269.688,A -85,B 0,C 180,E1 -16855.502,E2 -16855.502} C_VEL
LIN {X 0,Y 291.335,Z 269.695,A -85,B 0,C 180,E1 -16859.744,E2 -16859.744} C_VEL
LIN {X 0,Y 291.294,Z 269.7,A -85,B 0,C 180,E1 -16863.704,E2 -16863.704} C_VEL
LIN {X 0,Y 291.343,Z 269.692,A -85,B 0,C 180,E1 -16867.263,E2 -16867.263} C_VEL
LIN {X 0,Y 291.357,Z 269.691,A -85,B 0,C 180,E1 -16870.637,E2 -16870.637} C_VEL
LIN {X 0,Y 291.364,Z 269.69,A -85,B 0,C 180,E1 -16874.386,E2 -16874.386} C_VEL
LIN {X 0,Y 291.349,Z 269.692,A -85,B 0,C 180,E1 -16878.398,E2 -16878.398} C_VEL
LIN {X 0,Y 291.341,Z 269.693,A -85,B 0,C 180,E1 -16881.17,E2 -16881.17} C_VEL
LIN {X 0,Y 291.35,Z 269.691,A -85,B 0,C 180,E1 -16884.637,E2 -16884.637} C_VEL
LIN {X 0,Y 291.333,Z 269.695,A -85,B 0,C 180,E1 -16887.958,E2 -16887.958} C_VEL
LIN {X 0,Y 291.333,Z 269.696,A -85,B 0,C 180,E1 -16891.164,E2 -16891.164} C_VEL
LIN {X 0,Y 291.382,Z 269.685,A -85,B 0,C 180,E1 -16894.279,E2 -16894.279} C_VEL
LIN {X 0,Y 291.346,Z 269.695,A -85,B 0,C 180,E1 -16897.307,E2 -16897.307} C_VEL
LIN {X 0,Y 291.369,Z 269.685,A -85,B 0,C 180,E1 -16900.274,E2 -16900.274} C_VEL
LIN {X 0,Y 291.479,Z 269.675,A -85,B 0,C 180,E1 -16904.674,E2 -16904.674} C_VEL
LIN {X 0,Y 291.513,Z 269.674,A -85,B 0,C 180,E1 -16908.889,E2 -16908.889} C_VEL
LIN {X 0,Y 291.652,Z 269.653,A -85,B 0,C 180,E1 -16911.696,E2 -16911.696} C_VEL
LIN {X 0,Y 291.6,Z 269.661,A -85,B 0,C 180,E1 -16914.476,E2 -16914.476} C_VEL
LIN {X 0,Y 291.877,Z 269.616,A -85,B 0,C 180,E1 -16918.628,E2 -16918.628} C_VEL
LIN {X 0,Y 291.875,Z 269.625,A -85,B 0,C 180,E1 -16921.388,E2 -16921.388} C_VEL
LIN {X 0,Y 291.695,Z 269.651,A -85,B 0,C 180,E1 -16926.927,E2 -16926.927} C_VEL
LIN {X 0,Y 291.567,Z 269.665,A -85,B 0,C 180,E1 -16929.722,E2 -16929.722} C_VEL
LIN {X 0,Y 291.511,Z 269.673,A -85,B 0,C 180,E1 -16933.858,E2 -16933.858} C_VEL
LIN {X 0,Y 290.867,Z 269.756,A -85,B 0,C 180,E1 -16935.01,E2 -16935.01} C_VEL
LIN {X 0,Y 287.935,Z 270.118,A -85,B 0,C 180,E1 -16936.883,E2 -16936.883} C_VEL
LIN {X 0,Y 285.441,Z 270.432,A -85,B 0,C 180,E1 -16938.405,E2 -16938.405} C_VEL
LIN {X 0,Y 284.401,Z 270.558,A -85,B 0,C 180,E1 -16939.586,E2 -16939.586} C_VEL
LIN {X 0,Y 284.334,Z 270.568,A -85,B 0,C 180,E1 -16939.986,E2 -16939.986} C_VEL
LIN {X 0,Y 284.319,Z 270.57,A -85,B 0,C 180,E1 -16943.855,E2 -16943.855} C_VEL
LIN {X 0,Y 284.29,Z 270.574,A -85,B 0,C 180,E1 -16948.022,E2 -16948.022} C_VEL
LIN {X 0,Y 284.295,Z 270.575,A -85,B 0,C 180,E1 -16951.282,E2 -16951.282} C_VEL
LIN {X 0,Y 284.333,Z 270.852,A -85,B 0,C 180,E1 -16952.949,E2 -16952.949} C_VEL
LIN {X 0,Y 284.597,Z 272.775,A -85,B 0,C 180,E1 -16956.354,E2 -16956.354} C_VEL
LIN {X 0,Y 284.971,Z 275.131,A -85,B 0,C 180,E1 -16960.137,E2 -16960.137} C_VEL
LIN {X 0,Y 285.256,Z 277.516,A -85,B 0,C 180,E1 -16963.626,E2 -16963.626} C_VEL
LIN {X 0,Y 285.332,Z 279.57,A -85,B 0,C 180,E1 -16966.398,E2 -16966.398} C_VEL
LIN {X 0,Y 285.158,Z 282.305,A -85,B 0,C 180,E1 -16969.829,E2 -16969.829} C_VEL
LIN {X 0,Y 284.616,Z 285.603,A -85,B 0,C 180,E1 -16973.657,E2 -16973.657} C_VEL
LIN {X 0,Y 284.075,Z 288.859,A -85,B 0,C 180,E1 -16977.272,E2 -16977.272} C_VEL
LIN {X 0,Y 283.598,Z 291.697,A -85,B 0,C 180,E1 -16980.289,E2 -16980.289} C_VEL
LIN {X 0,Y 283.129,Z 295.357,A -85,B 0,C 180,E1 -16984.101,E2 -16984.101} C_VEL
LIN {X 0,Y 286.794,Z 309.502,A -85,B 0,C 180,E1 -16985.179,E2 -16985.179} C_VEL
LIN {X 0,Y 289.091,Z 320.653,A -85,B 0,C 180,E1 -16986.223,E2 -16986.223} C_VEL
LIN {X 0,Y 290.644,Z 332.521,A -85,B 0,C 180,E1 -16987.53,E2 -16987.53} C_VEL
LIN {X 0,Y 291.295,Z 341.113,A -85,B 0,C 180,E1 -16988.62,E2 -16988.62} C_VEL
LIN {X 0,Y 290.881,Z 346.371,A -85,B 0,C 180,E1 -16989.308,E2 -16989.308} C_VEL
LIN {X 0,Y 289.043,Z 356.514,A -85,B 0,C 180,E1 -16990.838,E2 -16990.838} C_VEL
LIN {X 0,Y 287.743,Z 364.349,A -85,B 0,C 180,E1 -16992.297,E2 -16992.297} C_VEL
LIN {X 0,Y 286.364,Z 371.856,A -85,B 0,C 180,E1 -16993.973,E2 -16993.973} C_VEL
LIN {X 0,Y 285.18,Z 378.394,A -85,B 0,C 180,E1 -16995.733,E2 -16995.733} C_VEL
LIN {X 0,Y 284.311,Z 382.894,A -85,B 0,C 180,E1 -16997.146,E2 -16997.146} C_VEL
LIN {X 0,Y 283.433,Z 388.389,A -85,B 0,C 180,E1 -16999.283,E2 -16999.283} C_VEL
LIN {X 0,Y 282.821,Z 392.716,A -85,B 0,C 180,E1 -17001.426,E2 -17001.426} C_VEL
LIN {X 0,Y 282.575,Z 395.085,A -85,B 0,C 180,E1 -17002.857,E2 -17002.857} C_VEL
LIN {X 0,Y 282.351,Z 397.394,A -85,B 0,C 180,E1 -17004.7,E2 -17004.7} C_VEL
LIN {X 0,Y 282.346,Z 399.337,A -85,B 0,C 180,E1 -17007.147,E2 -17007.147} C_VEL
LIN {X 0,Y 282.336,Z 399.927,A -85,B 0,C 180,E1 -17008.574,E2 -17008.574} C_VEL
LIN {X 0,Y 282.336,Z 399.927,A -85,B 0,C 180,E1 -17011.426,E2 -17011.426} C_VEL
LIN {X 0,Y 282.345,Z 399.337,A -85,B 0,C 180,E1 -17012.853,E2 -17012.853} C_VEL
LIN {X 0,Y 282.394,Z 396.886,A -85,B 0,C 180,E1 -17015.713,E2 -17015.713} C_VEL
LIN {X 0,Y 282.695,Z 393.934,A -85,B 0,C 180,E1 -17017.859,E2 -17017.859} C_VEL
LIN {X 0,Y 283.182,Z 389.943,A -85,B 0,C 180,E1 -17020.004,E2 -17020.004} C_VEL
LIN {X 0,Y 283.982,Z 384.811,A -85,B 0,C 180,E1 -17022.143,E2 -17022.143} C_VEL
LIN {X 0,Y 284.973,Z 379.55,A -85,B 0,C 180,E1 -17023.913,E2 -17023.913} C_VEL
LIN {X 0,Y 286.103,Z 373.232,A -85,B 0,C 180,E1 -17025.676,E2 -17025.676} C_VEL
LIN {X 0,Y 287.493,Z 365.952,A -85,B 0,C 180,E1 -17027.358,E2 -17027.358} C_VEL
LIN {X 0,Y 288.645,Z 358.432,A -85,B 0,C 180,E1 -17028.821,E2 -17028.821} C_VEL
LIN {X 0,Y 290.192,Z 349.906,A -85,B 0,C 180,E1 -17030.188,E2 -17030.188} C_VEL
LIN {X 0,Y 291.368,Z 342.313,A -85,B 0,C 180,E1 -17031.211,E2 -17031.211} C_VEL
LIN {X 0,Y 290.657,Z 332.668,A -85,B 0,C 180,E1 -17032.452,E2 -17032.452} C_VEL
LIN {X 0,Y 289.412,Z 322.437,A -85,B 0,C 180,E1 -17033.582,E2 -17033.582} C_VEL
LIN {X 0,Y 286.932,Z 310.145,A -85,B 0,C 180,E1 -17034.766,E2 -17034.766} C_VEL
LIN {X 0,Y 283.444,Z 297.245,A -85,B 0,C 180,E1 -17035.777,E2 -17035.777} C_VEL
LIN {X 0,Y 283.129,Z 295.364,A -85,B 0,C 180,E1 -17035.898,E2 -17035.898} C_VEL
LIN {X 0,Y 283.628,Z 291.499,A -85,B 0,C 180,E1 -17039.847,E2 -17039.847} C_VEL
LIN {X 0,Y 284.092,Z 288.599,A -85,B 0,C 180,E1 -17042.972,E2 -17042.972} C_VEL
LIN {X 0,Y 284.615,Z 285.563,A -85,B 0,C 180,E1 -17046.343,E2 -17046.343} C_VEL
LIN {X 0,Y 285.154,Z 282.304,A -85,B 0,C 180,E1 -17050.17,E2 -17050.17} C_VEL
LIN {X 0,Y 285.329,Z 279.56,A -85,B 0,C 180,E1 -17053.603,E2 -17053.603} C_VEL
LIN {X 0,Y 285.259,Z 277.512,A -85,B 0,C 180,E1 -17056.374,E2 -17056.374} C_VEL
LIN {X 0,Y 284.94,Z 274.971,A -85,B 0,C 180,E1 -17060.104,E2 -17060.104} C_VEL
LIN {X 0,Y 284.596,Z 272.775,A -85,B 0,C 180,E1 -17063.646,E2 -17063.646} C_VEL
LIN {X 0,Y 284.327,Z 270.782,A -85,B 0,C 180,E1 -17067.182,E2 -17067.182} C_VEL
LIN {X 0,Y 284.346,Z 270.568,A -85,B 0,C 180,E1 -17070.367,E2 -17070.367} C_VEL
LIN {X 0,Y 284.308,Z 270.572,A -85,B 0,C 180,E1 -17073.572,E2 -17073.572} C_VEL
LIN {X 0,Y 284.328,Z 270.568,A -85,B 0,C 180,E1 -17076.696,E2 -17076.696} C_VEL
LIN {X 0,Y 284.337,Z 270.567,A -85,B 0,C 180,E1 -17081.25,E2 -17081.25} C_VEL
LIN {X 0,Y 284.465,Z 270.553,A -85,B 0,C 180,E1 -17085.689,E2 -17085.689} C_VEL
LIN {X 0,Y 284.513,Z 270.544,A -85,B 0,C 180,E1 -17090.035,E2 -17090.035} C_VEL
LIN {X 0,Y 284.65,Z 270.527,A -85,B 0,C 180,E1 -17092.901,E2 -17092.901} C_VEL
LIN {X 0,Y 284.841,Z 270.501,A -85,B 0,C 180,E1 -17098.578,E2 -17098.578} C_VEL
LIN {X 0,Y 284.844,Z 270.49,A -85,B 0,C 180,E1 -17101.405,E2 -17101.405} C_VEL
LIN {X 0,Y 284.645,Z 270.53,A -85,B 0,C 180,E1 -17107.083,E2 -17107.083} C_VEL
LIN {X 0,Y 284.499,Z 270.542,A -85,B 0,C 180,E1 -17109.949,E2 -17109.949} C_VEL
LIN {X 0,Y 284.445,Z 270.55,A -85,B 0,C 180,E1 -17114.295,E2 -17114.295} C_VEL
LIN {X 0,Y 284.311,Z 270.57,A -85,B 0,C 180,E1 -17118.735,E2 -17118.735} C_VEL
LIN {X 0,Y 284.307,Z 270.568,A -85,B 0,C 180,E1 -17123.288,E2 -17123.288} C_VEL
LIN {X 0,Y 284.362,Z 270.562,A -85,B 0,C 180,E1 -17127.162,E2 -17127.162} C_VEL
LIN {X 0,Y 284.255,Z 270.575,A -85,B 0,C 180,E1 -17131.267,E2 -17131.267} C_VEL
LIN {X 0,Y 284.327,Z 270.566,A -85,B 0,C 180,E1 -17135.346,E2 -17135.346} C_VEL
LIN {X 0,Y 284.294,Z 270.573,A -85,B 0,C 180,E1 -17138.159,E2 -17138.159} C_VEL
LIN {X 0,Y 284.304,Z 270.573,A -85,B 0,C 180,E1 -17142.134,E2 -17142.134} C_VEL
LIN {X 0,Y 284.31,Z 270.572,A -85,B 0,C 180,E1 -17146.201,E2 -17146.201} C_VEL
LIN {X 0,Y 284.307,Z 270.572,A -85,B 0,C 180,E1 -17150.007,E2 -17150.007} C_VEL
LIN {X 0,Y 284.299,Z 270.572,A -85,B 0,C 180,E1 -17153.61,E2 -17153.61} C_VEL
LIN {X 0,Y 284.258,Z 270.576,A -85,B 0,C 180,E1 -17157.184,E2 -17157.184} C_VEL
LIN {X 0,Y 284.307,Z 270.57,A -85,B 0,C 180,E1 -17160.371,E2 -17160.371} C_VEL
LIN {X 0,Y 284.332,Z 270.569,A -85,B 0,C 180,E1 -17163.886,E2 -17163.886} C_VEL
LIN {X 0,Y 285.346,Z 273.414,A -85,B 0,C 180,E1 -17164.068,E2 -17164.068} C_VEL
LIN {X 0,Y 291.741,Z 286.596,A -85,B 0,C 180,E1 -17165.156,E2 -17165.156} C_VEL
LIN {X 0,Y 297.366,Z 295.978,A -85,B 0,C 180,E1 -17166.191,E2 -17166.191} C_VEL
LIN {X 0,Y 304.31,Z 305.426,A -85,B 0,C 180,E1 -17167.458,E2 -17167.458} C_VEL
LIN {X 0,Y 311.754,Z 314.557,A -85,B 0,C 180,E1 -17168.858,E2 -17168.858} C_VEL
LIN {X 0,Y 319.159,Z 322.868,A -85,B 0,C 180,E1 -17170.394,E2 -17170.394} C_VEL
LIN {X 0,Y 325.377,Z 329.484,A -85,B 0,C 180,E1 -17171.841,E2 -17171.841} C_VEL
LIN {X 0,Y 331.793,Z 336.022,A -85,B 0,C 180,E1 -17173.474,E2 -17173.474} C_VEL
LIN {X 0,Y 337.315,Z 341.413,A -85,B 0,C 180,E1 -17175.062,E2 -17175.062} C_VEL
LIN {X 0,Y 341.223,Z 344.869,A -85,B 0,C 180,E1 -17176.269,E2 -17176.269} C_VEL
LIN {X 0,Y 346.878,Z 350.14,A -85,B 0,C 180,E1 -17178.311,E2 -17178.311} C_VEL
LIN {X 0,Y 350.28,Z 352.652,A -85,B 0,C 180,E1 -17179.597,E2 -17179.597} C_VEL
LIN {X 0,Y 352.841,Z 354.893,A -85,B 0,C 180,E1 -17180.831,E2 -17180.831} C_VEL
LIN {X 0,Y 354.874,Z 356.948,A -85,B 0,C 180,E1 -17182.032,E2 -17182.032} C_VEL
LIN {X 0,Y 356.746,Z 358.546,A -85,B 0,C 180,E1 -17183.212,E2 -17183.212} C_VEL
LIN {X 0,Y 359.593,Z 360.395,A -85,B 0,C 180,E1 -17185.264,E2 -17185.264} C_VEL
LIN {X 0,Y 361.233,Z 361.041,A -85,B 0,C 180,E1 -17186.654,E2 -17186.654} C_VEL
LIN {X 0,Y 362.233,Z 361.34,A -85,B 0,C 180,E1 -17187.776,E2 -17187.776} C_VEL
LIN {X 0,Y 362.866,Z 361.479,A -85,B 0,C 180,E1 -17188.89,E2 -17188.89} C_VEL
LIN {X 0,Y 363.084,Z 361.518,A -85,B 0,C 180,E1 -17190,E2 -17190} C_VEL
LIN {X 0,Y 362.865,Z 361.481,A -85,B 0,C 180,E1 -17191.11,E2 -17191.11} C_VEL
LIN {X 0,Y 362.226,Z 361.343,A -85,B 0,C 180,E1 -17192.224,E2 -17192.224} C_VEL
LIN {X 0,Y 361.211,Z 361.054,A -85,B 0,C 180,E1 -17193.346,E2 -17193.346} C_VEL
LIN {X 0,Y 359.599,Z 360.383,A -85,B 0,C 180,E1 -17194.749,E2 -17194.749} C_VEL
LIN {X 0,Y 356.716,Z 358.556,A -85,B 0,C 180,E1 -17196.789,E2 -17196.789} C_VEL
LIN {X 0,Y 354.805,Z 356.861,A -85,B 0,C 180,E1 -17198.018,E2 -17198.018} C_VEL
LIN {X 0,Y 352.035,Z 354.041,A -85,B 0,C 180,E1 -17199.618,E2 -17199.618} C_VEL
LIN {X 0,Y 348.608,Z 351.486,A -85,B 0,C 180,E1 -17201.025,E2 -17201.025} C_VEL
LIN {X 0,Y 343.358,Z 346.809,A -85,B 0,C 180,E1 -17203.012,E2 -17203.012} C_VEL
LIN {X 0,Y 337.525,Z 341.564,A -85,B 0,C 180,E1 -17204.884,E2 -17204.884} C_VEL
LIN {X 0,Y 331.812,Z 335.998,A -85,B 0,C 180,E1 -17206.523,E2 -17206.523} C_VEL
LIN {X 0,Y 325.384,Z 329.497,A -85,B 0,C 180,E1 -17208.163,E2 -17208.163} C_VEL
LIN {X 0,Y 318.002,Z 321.658,A -85,B 0,C 180,E1 -17209.845,E2 -17209.845} C_VEL
LIN {X 0,Y 311.191,Z 313.849,A -85,B 0,C 180,E1 -17211.256,E2 -17211.256} C_VEL
LIN {X 0,Y 302.964,Z 303.695,A -85,B 0,C 180,E1 -17212.793,E2 -17212.793} C_VEL
LIN {X 0,Y 295.718,Z 293.414,A -85,B 0,C 180,E1 -17214.117,E2 -17214.117} C_VEL
LIN {X 0,Y 290.415,Z 284.093,A -85,B 0,C 180,E1 -17215.075,E2 -17215.075} C_VEL
LIN {X 0,Y 284.425,Z 271.18,A -85,B 0,C 180,E1 -17216.084,E2 -17216.084} C_VEL
LIN {X 0,Y 284.338,Z 270.568,A -85,B 0,C 180,E1 -17216.14,E2 -17216.14} C_VEL
LIN {X 0,Y 284.263,Z 270.578,A -85,B 0,C 180,E1 -17220.103,E2 -17220.103} C_VEL
LIN {X 0,Y 284.256,Z 270.576,A -85,B 0,C 180,E1 -17222.951,E2 -17222.951} C_VEL
LIN {X 0,Y 284.299,Z 270.572,A -85,B 0,C 180,E1 -17226.39,E2 -17226.39} C_VEL
LIN {X 0,Y 284.307,Z 270.572,A -85,B 0,C 180,E1 -17229.993,E2 -17229.993} C_VEL
LIN {X 0,Y 284.314,Z 270.569,A -85,B 0,C 180,E1 -17234.22,E2 -17234.22} C_VEL
LIN {X 0,Y 284.301,Z 270.571,A -85,B 0,C 180,E1 -17238.144,E2 -17238.144} C_VEL
LIN {X 0,Y 284.303,Z 270.57,A -85,B 0,C 180,E1 -17242.281,E2 -17242.281} C_VEL
LIN {X 0,Y 284.289,Z 270.573,A -85,B 0,C 180,E1 -17245.361,E2 -17245.361} C_VEL
LIN {X 0,Y 284.255,Z 270.575,A -85,B 0,C 180,E1 -17248.733,E2 -17248.733} C_VEL
LIN {X 0,Y 284.362,Z 270.562,A -85,B 0,C 180,E1 -17252.838,E2 -17252.838} C_VEL
LIN {X 0,Y 284.307,Z 270.568,A -85,B 0,C 180,E1 -17256.712,E2 -17256.712} C_VEL
LIN {X 0,Y 284.311,Z 270.57,A -85,B 0,C 180,E1 -17261.265,E2 -17261.265} C_VEL
LIN {X 0,Y 284.445,Z 270.55,A -85,B 0,C 180,E1 -17265.705,E2 -17265.705} C_VEL
LIN {X 0,Y 284.499,Z 270.542,A -85,B 0,C 180,E1 -17270.051,E2 -17270.051} C_VEL
LIN {X 0,Y 284.645,Z 270.53,A -85,B 0,C 180,E1 -17272.917,E2 -17272.917} C_VEL
LIN {X 0,Y 284.844,Z 270.49,A -85,B 0,C 180,E1 -17278.595,E2 -17278.595} C_VEL
LIN {X 0,Y 284.841,Z 270.501,A -85,B 0,C 180,E1 -17281.422,E2 -17281.422} C_VEL
LIN {X 0,Y 284.65,Z 270.527,A -85,B 0,C 180,E1 -17287.099,E2 -17287.099} C_VEL
LIN {X 0,Y 284.513,Z 270.544,A -85,B 0,C 180,E1 -17289.965,E2 -17289.965} C_VEL
LIN {X 0,Y 284.465,Z 270.554,A -85,B 0,C 180,E1 -17294.311,E2 -17294.311} C_VEL
LIN {X 0,Y 284.337,Z 270.566,A -85,B 0,C 180,E1 -17298.75,E2 -17298.75} C_VEL
LIN {X 0,Y 284.334,Z 270.568,A -85,B 0,C 180,E1 -17299.986,E2 -17299.986} C_VEL
LIN {X 0,Y 283.703,Z 270.652,A -85,B 0,C 180,E1 -17301.169,E2 -17301.169} C_VEL
LIN {X 0,Y 280.819,Z 271.012,A -85,B 0,C 180,E1 -17303.095,E2 -17303.095} C_VEL
LIN {X 0,Y 278.357,Z 271.314,A -85,B 0,C 180,E1 -17304.659,E2 -17304.659} C_VEL
LIN {X 0,Y 277.317,Z 271.444,A -85,B 0,C 180,E1 -17305.873,E2 -17305.873} C_VEL
LIN {X 0,Y 277.243,Z 271.447,A -85,B 0,C 180,E1 -17306.284,E2 -17306.284} C_VEL
LIN {X 0,Y 277.259,Z 271.451,A -85,B 0,C 180,E1 -17310.479,E2 -17310.479} C_VEL
LIN {X 0,Y 277.256,Z 271.557,A -85,B 0,C 180,E1 -17312.17,E2 -17312.17} C_VEL
LIN {X 0,Y 277.543,Z 273.568,A -85,B 0,C 180,E1 -17315.876,E2 -17315.876} C_VEL
LIN {X 0,Y 277.832,Z 275.586,A -85,B 0,C 180,E1 -17319.235,E2 -17319.235} C_VEL
LIN {X 0,Y 278.183,Z 278.061,A -85,B 0,C 180,E1 -17323.018,E2 -17323.018} C_VEL
LIN {X 0,Y 278.311,Z 279.455,A -85,B 0,C 180,E1 -17325.005,E2 -17325.005} C_VEL
LIN {X 0,Y 278.176,Z 282.45,A -85,B 0,C 180,E1 -17328.939,E2 -17328.939} C_VEL
LIN {X 0,Y 277.71,Z 285.472,A -85,B 0,C 180,E1 -17332.602,E2 -17332.602} C_VEL
LIN {X 0,Y 277.147,Z 288.485,A -85,B 0,C 180,E1 -17336.091,E2 -17336.091} C_VEL
LIN {X 0,Y 276.615,Z 291.824,A -85,B 0,C 180,E1 -17339.762,E2 -17339.762} C_VEL
LIN {X 0,Y 276.139,Z 295.266,A -85,B 0,C 180,E1 -17343.422,E2 -17343.422} C_VEL
LIN {X 0,Y 277.69,Z 301.035,A -85,B 0,C 180,E1 -17343.833,E2 -17343.833} C_VEL
LIN {X 0,Y 280.49,Z 312.099,A -85,B 0,C 180,E1 -17344.79,E2 -17344.79} C_VEL
LIN {X 0,Y 282.583,Z 322.825,A -85,B 0,C 180,E1 -17345.869,E2 -17345.869} C_VEL
LIN {X 0,Y 283.781,Z 332.317,A -85,B 0,C 180,E1 -17346.956,E2 -17346.956} C_VEL
LIN {X 0,Y 284.468,Z 341.015,A -85,B 0,C 180,E1 -17348.095,E2 -17348.095} C_VEL
LIN {X 0,Y 284.429,Z 344.824,A -85,B 0,C 180,E1 -17348.626,E2 -17348.626} C_VEL
LIN {X 0,Y 282.352,Z 356.319,A -85,B 0,C 180,E1 -17350.365,E2 -17350.365} C_VEL
LIN {X 0,Y 280.788,Z 364.953,A -85,B 0,C 180,E1 -17352.028,E2 -17352.028} C_VEL
LIN {X 0,Y 279.521,Z 371.661,A -85,B 0,C 180,E1 -17353.57,E2 -17353.57} C_VEL
LIN {X 0,Y 278.285,Z 378.199,A -85,B 0,C 180,E1 -17355.372,E2 -17355.372} C_VEL
LIN {X 0,Y 277.364,Z 382.699,A -85,B 0,C 180,E1 -17356.818,E2 -17356.818} C_VEL
LIN {X 0,Y 276.418,Z 388.193,A -85,B 0,C 180,E1 -17359.007,E2 -17359.007} C_VEL
LIN {X 0,Y 275.761,Z 392.52,A -85,B 0,C 180,E1 -17361.204,E2 -17361.204} C_VEL
LIN {X 0,Y 275.515,Z 394.89,A -85,B 0,C 180,E1 -17362.673,E2 -17362.673} C_VEL
LIN {X 0,Y 275.245,Z 397.433,A -85,B 0,C 180,E1 -17364.809,E2 -17364.809} C_VEL
LIN {X 0,Y 275.255,Z 399.143,A -85,B 0,C 180,E1 -17367.073,E2 -17367.073} C_VEL
LIN {X 0,Y 275.262,Z 399.733,A -85,B 0,C 180,E1 -17368.537,E2 -17368.537} C_VEL
LIN {X 0,Y 275.262,Z 399.733,A -85,B 0,C 180,E1 -17371.463,E2 -17371.463} C_VEL
LIN {X 0,Y 275.254,Z 399.143,A -85,B 0,C 180,E1 -17372.927,E2 -17372.927} C_VEL
LIN {X 0,Y 275.314,Z 396.691,A -85,B 0,C 180,E1 -17375.86,E2 -17375.86} C_VEL
LIN {X 0,Y 275.623,Z 393.739,A -85,B 0,C 180,E1 -17378.062,E2 -17378.062} C_VEL
LIN {X 0,Y 276.175,Z 389.748,A -85,B 0,C 180,E1 -17380.261,E2 -17380.261} C_VEL
LIN {X 0,Y 277.004,Z 384.615,A -85,B 0,C 180,E1 -17382.454,E2 -17382.454} C_VEL
LIN {X 0,Y 278.038,Z 379.354,A -85,B 0,C 180,E1 -17384.267,E2 -17384.267} C_VEL
LIN {X 0,Y 279.238,Z 373.036,A -85,B 0,C 180,E1 -17386.072,E2 -17386.072} C_VEL
LIN {X 0,Y 280.569,Z 366.442,A -85,B 0,C 180,E1 -17387.642,E2 -17387.642} C_VEL
LIN {X 0,Y 281.926,Z 358.237,A -85,B 0,C 180,E1 -17389.287,E2 -17389.287} C_VEL
LIN {X 0,Y 283.542,Z 349.711,A -85,B 0,C 180,E1 -17390.683,E2 -17390.683} C_VEL
LIN {X 0,Y 284.552,Z 343.47,A -85,B 0,C 180,E1 -17391.554,E2 -17391.554} C_VEL
LIN {X 0,Y 284.036,Z 335.077,A -85,B 0,C 180,E1 -17392.699,E2 -17392.699} C_VEL
LIN {X 0,Y 282.973,Z 325.204,A -85,B 0,C 180,E1 -17393.867,E2 -17393.867} C_VEL
LIN {X 0,Y 281.287,Z 315.734,A -85,B 0,C 180,E1 -17394.858,E2 -17394.858} C_VEL
LIN {X 0,Y 278.81,Z 305.32,A -85,B 0,C 180,E1 -17395.811,E2 -17395.811} C_VEL
LIN {X 0,Y 276.133,Z 295.171,A -85,B 0,C 180,E1 -17396.628,E2 -17396.628} C_VEL
LIN {X 0,Y 276.643,Z 291.455,A -85,B 0,C 180,E1 -17400.536,E2 -17400.536} C_VEL
LIN {X 0,Y 277.141,Z 288.443,A -85,B 0,C 180,E1 -17403.91,E2 -17403.91} C_VEL
LIN {X 0,Y 277.709,Z 285.43,A -85,B 0,C 180,E1 -17407.398,E2 -17407.398} C_VEL
LIN {X 0,Y 278.16,Z 282.434,A -85,B 0,C 180,E1 -17411.064,E2 -17411.064} C_VEL
LIN {X 0,Y 278.311,Z 279.451,A -85,B 0,C 180,E1 -17414.995,E2 -17414.995} C_VEL
LIN {X 0,Y 278.032,Z 276.76,A -85,B 0,C 180,E1 -17418.904,E2 -17418.904} C_VEL
LIN {X 0,Y 277.664,Z 274.467,A -85,B 0,C 180,E1 -17422.585,E2 -17422.585} C_VEL
LIN {X 0,Y 277.348,Z 272.126,A -85,B 0,C 180,E1 -17426.741,E2 -17426.741} C_VEL
LIN {X 0,Y 277.256,Z 271.56,A -85,B 0,C 180,E1 -17427.83,E2 -17427.83} C_VEL
LIN {X 0,Y 277.248,Z 271.451,A -85,B 0,C 180,E1 -17431.2,E2 -17431.2} C_VEL
LIN {X 0,Y 277.247,Z 271.45,A -85,B 0,C 180,E1 -17434.465,E2 -17434.465} C_VEL
LIN {X 0,Y 277.264,Z 271.451,A -85,B 0,C 180,E1 -17437.645,E2 -17437.645} C_VEL
LIN {X 0,Y 277.29,Z 271.444,A -85,B 0,C 180,E1 -17440.755,E2 -17440.755} C_VEL
LIN {X 0,Y 277.412,Z 271.43,A -85,B 0,C 180,E1 -17445.317,E2 -17445.317} C_VEL
LIN {X 0,Y 277.455,Z 271.424,A -85,B 0,C 180,E1 -17449.779,E2 -17449.779} C_VEL
LIN {X 0,Y 277.608,Z 271.404,A -85,B 0,C 180,E1 -17452.72,E2 -17452.72} C_VEL
LIN {X 0,Y 277.807,Z 271.377,A -85,B 0,C 180,E1 -17458.542,E2 -17458.542} C_VEL
LIN {X 0,Y 277.81,Z 271.365,A -85,B 0,C 180,E1 -17461.441,E2 -17461.441} C_VEL
LIN {X 0,Y 277.602,Z 271.406,A -85,B 0,C 180,E1 -17467.263,E2 -17467.263} C_VEL
LIN {X 0,Y 277.44,Z 271.421,A -85,B 0,C 180,E1 -17470.205,E2 -17470.205} C_VEL
LIN {X 0,Y 277.391,Z 271.43,A -85,B 0,C 180,E1 -17474.667,E2 -17474.667} C_VEL
LIN {X 0,Y 277.263,Z 271.443,A -85,B 0,C 180,E1 -17479.229,E2 -17479.229} C_VEL
LIN {X 0,Y 277.271,Z 271.444,A -85,B 0,C 180,E1 -17483.915,E2 -17483.915} C_VEL
LIN {X 0,Y 277.289,Z 271.443,A -85,B 0,C 180,E1 -17487.493,E2 -17487.493} C_VEL
LIN {X 0,Y 277.217,Z 271.455,A -85,B 0,C 180,E1 -17490.464,E2 -17490.464} C_VEL
LIN {X 0,Y 277.22,Z 271.451,A -85,B 0,C 180,E1 -17493.887,E2 -17493.887} C_VEL
LIN {X 0,Y 277.249,Z 271.448,A -85,B 0,C 180,E1 -17497.459,E2 -17497.459} C_VEL
LIN {X 0,Y 277.227,Z 271.451,A -85,B 0,C 180,E1 -17501.219,E2 -17501.219} C_VEL
LIN {X 0,Y 277.246,Z 271.447,A -85,B 0,C 180,E1 -17505.201,E2 -17505.201} C_VEL
LIN {X 0,Y 277.251,Z 271.448,A -85,B 0,C 180,E1 -17509.488,E2 -17509.488} C_VEL
LIN {X 0,Y 277.235,Z 271.451,A -85,B 0,C 180,E1 -17512.527,E2 -17512.527} C_VEL
LIN {X 0,Y 277.205,Z 271.457,A -85,B 0,C 180,E1 -17516.099,E2 -17516.099} C_VEL
LIN {X 0,Y 277.212,Z 271.456,A -85,B 0,C 180,E1 -17519.533,E2 -17519.533} C_VEL
LIN {X 0,Y 277.305,Z 271.444,A -85,B 0,C 180,E1 -17523.174,E2 -17523.174} C_VEL
